LIN {X 0,Y 249.266,Z 167.431,A -85,B 0,C 180,E1 -18895.147,E2 -18895.147} C_VEL
LIN {X 0,Y 249.661,Z 167.386,A -85,B 0,C 180,E1 -18898.386,E2 -18898.386} C_VEL
LIN {X 0,Y 249.66,Z 167.377,A -85,B 0,C 180,E1 -18901.612,E2 -18901.612} C_VEL
LIN {X 0,Y 249.426,Z 167.411,A -85,B 0,C 180,E1 -18906.555,E2 -18906.555} C_VEL
LIN {X 0,Y 249.335,Z 167.427,A -85,B 0,C 180,E1 -18909.735,E2 -18909.735} C_VEL
LIN {X 0,Y 249.147,Z 167.433,A -85,B 0,C 180,E1 -18914.705,E2 -18914.705} C_VEL
LIN {X 0,Y 249.08,Z 167.45,A -85,B 0,C 180,E1 -18918.08,E2 -18918.08} C_VEL
LIN {X 0,Y 249.043,Z 167.464,A -85,B 0,C 180,E1 -18921.521,E2 -18921.521} C_VEL
LIN {X 0,Y 249.043,Z 167.454,A -85,B 0,C 180,E1 -18925.438,E2 -18925.438} C_VEL
LIN {X 0,Y 249.023,Z 167.452,A -85,B 0,C 180,E1 -18928.967,E2 -18928.967} C_VEL
LIN {X 0,Y 249.025,Z 167.464,A -85,B 0,C 180,E1 -18932.425,E2 -18932.425} C_VEL
LIN {X 0,Y 249.008,Z 167.459,A -85,B 0,C 180,E1 -18936.347,E2 -18936.347} C_VEL
LIN {X 0,Y 248.979,Z 167.466,A -85,B 0,C 180,E1 -18940.481,E2 -18940.481} C_VEL
LIN {X 0,Y 248.959,Z 167.473,A -85,B 0,C 180,E1 -18944.887,E2 -18944.887} C_VEL
LIN {X 0,Y 248.975,Z 167.462,A -85,B 0,C 180,E1 -18947.353,E2 -18947.353} C_VEL
LIN {X 0,Y 249.036,Z 167.465,A -85,B 0,C 180,E1 -18952.2,E2 -18952.2} C_VEL
LIN {X 0,Y 249.038,Z 167.459,A -85,B 0,C 180,E1 -18955.638,E2 -18955.638} C_VEL
LIN {X 0,Y 248.997,Z 167.467,A -85,B 0,C 180,E1 -18959.465,E2 -18959.465} C_VEL
LIN {X 0,Y 249.016,Z 167.467,A -85,B 0,C 180,E1 -18963.155,E2 -18963.155} C_VEL
LIN {X 0,Y 249,Z 167.461,A -85,B 0,C 180,E1 -18966.724,E2 -18966.724} C_VEL
LIN {X 0,Y 249.037,Z 167.466,A -85,B 0,C 180,E1 -18970.205,E2 -18970.205} C_VEL
LIN {X 0,Y 249.152,Z 167.449,A -85,B 0,C 180,E1 -18973.615,E2 -18973.615} C_VEL
LIN {X 0,Y 249.214,Z 167.439,A -85,B 0,C 180,E1 -18978.614,E2 -18978.614} C_VEL
LIN {X 0,Y 249.355,Z 167.424,A -85,B 0,C 180,E1 -18980.552,E2 -18980.552} C_VEL
LIN {X 0,Y 250.451,Z 170.4,A -85,B 0,C 180,E1 -18980.803,E2 -18980.803} C_VEL
LIN {X 0,Y 254.125,Z 177.882,A -85,B 0,C 180,E1 -18981.488,E2 -18981.488} C_VEL
LIN {X 0,Y 263.092,Z 200.069,A -85,B 0,C 180,E1 -18983.19,E2 -18983.19} C_VEL
LIN {X 0,Y 264.812,Z 205.047,A -85,B 0,C 180,E1 -18983.523,E2 -18983.523} C_VEL
LIN {X 0,Y 262.363,Z 274.189,A -85,B 0,C 180,E1 -18985.433,E2 -18985.433} C_VEL
LIN {X 0,Y 261.405,Z 287.63,A -85,B 0,C 180,E1 -18986.1,E2 -18986.1} C_VEL
LIN {X 0,Y 260.23,Z 300.609,A -85,B 0,C 180,E1 -18987.077,E2 -18987.077} C_VEL
LIN {X 0,Y 258.83,Z 312.038,A -85,B 0,C 180,E1 -18988.249,E2 -18988.249} C_VEL
LIN {X 0,Y 257.009,Z 323.786,A -85,B 0,C 180,E1 -18989.804,E2 -18989.804} C_VEL
LIN {X 0,Y 255.145,Z 334.352,A -85,B 0,C 180,E1 -18991.578,E2 -18991.578} C_VEL
LIN {X 0,Y 253.465,Z 343.314,A -85,B 0,C 180,E1 -18993.467,E2 -18993.467} C_VEL
LIN {X 0,Y 251.739,Z 351.564,A -85,B 0,C 180,E1 -18995.607,E2 -18995.607} C_VEL
LIN {X 0,Y 250.15,Z 359.176,A -85,B 0,C 180,E1 -18998.075,E2 -18998.075} C_VEL
LIN {X 0,Y 248.942,Z 365.251,A -85,B 0,C 180,E1 -19000.574,E2 -19000.574} C_VEL
LIN {X 0,Y 248.007,Z 370.011,A -85,B 0,C 180,E1 -19003.103,E2 -19003.103} C_VEL
LIN {X 0,Y 247.471,Z 372.881,A -85,B 0,C 180,E1 -19005.084,E2 -19005.084} C_VEL
LIN {X 0,Y 247.146,Z 374.563,A -85,B 0,C 180,E1 -19006.521,E2 -19006.521} C_VEL
LIN {X 0,Y 246.896,Z 376.129,A -85,B 0,C 180,E1 -19008.247,E2 -19008.247} C_VEL
LIN {X 0,Y 246.775,Z 377.22,A -85,B 0,C 180,E1 -19009.983,E2 -19009.983} C_VEL
LIN {X 0,Y 246.672,Z 377.893,A -85,B 0,C 180,E1 -19011.739,E2 -19011.739} C_VEL
LIN {X 0,Y 246.81,Z 378.021,A -85,B 0,C 180,E1 -19014.331,E2 -19014.331} C_VEL
LIN {X 0,Y 247.173,Z 377.088,A -85,B 0,C 180,E1 -19017.061,E2 -19017.061} C_VEL
LIN {X 0,Y 247.576,Z 375.846,A -85,B 0,C 180,E1 -19018.854,E2 -19018.854} C_VEL
LIN {X 0,Y 248.6,Z 372.467,A -85,B 0,C 180,E1 -19021.996,E2 -19021.996} C_VEL
LIN {X 0,Y 250.01,Z 367.842,A -85,B 0,C 180,E1 -19024.887,E2 -19024.887} C_VEL
LIN {X 0,Y 251.599,Z 362.394,A -85,B 0,C 180,E1 -19027.412,E2 -19027.412} C_VEL
LIN {X 0,Y 253.768,Z 354.935,A -85,B 0,C 180,E1 -19030.083,E2 -19030.083} C_VEL
LIN {X 0,Y 255.796,Z 347.755,A -85,B 0,C 180,E1 -19032.115,E2 -19032.115} C_VEL
LIN {X 0,Y 258.174,Z 338.472,A -85,B 0,C 180,E1 -19034.232,E2 -19034.232} C_VEL
LIN {X 0,Y 260.745,Z 327.432,A -85,B 0,C 180,E1 -19036.205,E2 -19036.205} C_VEL
LIN {X 0,Y 262.8,Z 317.371,A -85,B 0,C 180,E1 -19037.626,E2 -19037.626} C_VEL
LIN {X 0,Y 264.715,Z 306.116,A -85,B 0,C 180,E1 -19038.88,E2 -19038.88} C_VEL
LIN {X 0,Y 266.377,Z 293.716,A -85,B 0,C 180,E1 -19039.918,E2 -19039.918} C_VEL
LIN {X 0,Y 267.556,Z 280.481,A -85,B 0,C 180,E1 -19040.713,E2 -19040.713} C_VEL
LIN {X 0,Y 268.409,Z 267.04,A -85,B 0,C 180,E1 -19041.175,E2 -19041.175} C_VEL
LIN {X 0,Y 270.741,Z 210.533,A -85,B 0,C 180,E1 -19042.703,E2 -19042.703} C_VEL
LIN {X 0,Y 264.124,Z 195.268,A -85,B 0,C 180,E1 -19044.23,E2 -19044.23} C_VEL
LIN {X 0,Y 256.806,Z 181.169,A -85,B 0,C 180,E1 -19045.966,E2 -19045.966} C_VEL
LIN {X 0,Y 250.919,Z 171.414,A -85,B 0,C 180,E1 -19047.421,E2 -19047.421} C_VEL
LIN {X 0,Y 249.354,Z 168.806,A -85,B 0,C 180,E1 -19047.828,E2 -19047.828} C_VEL
LIN {X 0,Y 249.187,Z 168.189,A -85,B 0,C 180,E1 -19048.008,E2 -19048.008} C_VEL
LIN {X 0,Y 249.045,Z 167.461,A -85,B 0,C 180,E1 -19048.395,E2 -19048.395} C_VEL
LIN {X 0,Y 249.095,Z 167.458,A -85,B 0,C 180,E1 -19051.34,E2 -19051.34} C_VEL
LIN {X 0,Y 249.15,Z 167.451,A -85,B 0,C 180,E1 -19054.97,E2 -19054.97} C_VEL
LIN {X 0,Y 249.103,Z 167.456,A -85,B 0,C 180,E1 -19060.212,E2 -19060.212} C_VEL
LIN {X 0,Y 249.195,Z 167.44,A -85,B 0,C 180,E1 -19063.62,E2 -19063.62} C_VEL
LIN {X 0,Y 249.241,Z 167.438,A -85,B 0,C 180,E1 -19068.617,E2 -19068.617} C_VEL
LIN {X 0,Y 249.436,Z 167.403,A -85,B 0,C 180,E1 -19071.903,E2 -19071.903} C_VEL
LIN {X 0,Y 249.296,Z 167.415,A -85,B 0,C 180,E1 -19075.507,E2 -19075.507} C_VEL
LIN {X 0,Y 249.673,Z 167.382,A -85,B 0,C 180,E1 -19078.388,E2 -19078.388} C_VEL
LIN {X 0,Y 249.663,Z 167.37,A -85,B 0,C 180,E1 -19081.614,E2 -19081.614} C_VEL
LIN {X 0,Y 249.489,Z 167.394,A -85,B 0,C 180,E1 -19082.511,E2 -19082.511} C_VEL
LIN {X 0,Y 248.709,Z 167.502,A -85,B 0,C 180,E1 -19083.857,E2 -19083.857} C_VEL
LIN {X 0,Y 245.911,Z 167.861,A -85,B 0,C 180,E1 -19086.056,E2 -19086.056} C_VEL
LIN {X 0,Y 242.72,Z 168.25,A -85,B 0,C 180,E1 -19088.763,E2 -19088.763} C_VEL
LIN {X 0,Y 242.313,Z 168.291,A -85,B 0,C 180,E1 -19089.698,E2 -19089.698} C_VEL
LIN {X 0,Y 242.119,Z 168.317,A -85,B 0,C 180,E1 -19095.145,E2 -19095.145} C_VEL
LIN {X 0,Y 242.031,Z 168.337,A -85,B 0,C 180,E1 -19098.629,E2 -19098.629} C_VEL
LIN {X 0,Y 241.975,Z 168.332,A -85,B 0,C 180,E1 -19102.185,E2 -19102.185} C_VEL
LIN {X 0,Y 241.989,Z 168.329,A -85,B 0,C 180,E1 -19105.827,E2 -19105.827} C_VEL
LIN {X 0,Y 241.971,Z 168.337,A -85,B 0,C 180,E1 -19109.59,E2 -19109.59} C_VEL
LIN {X 0,Y 241.982,Z 168.338,A -85,B 0,C 180,E1 -19113.494,E2 -19113.494} C_VEL
LIN {X 0,Y 241.967,Z 168.338,A -85,B 0,C 180,E1 -19117.587,E2 -19117.587} C_VEL
LIN {X 0,Y 241.907,Z 168.352,A -85,B 0,C 180,E1 -19121.93,E2 -19121.93} C_VEL
LIN {X 0,Y 241.902,Z 168.356,A -85,B 0,C 180,E1 -19126.581,E2 -19126.581} C_VEL
LIN {X 0,Y 241.927,Z 168.36,A -85,B 0,C 180,E1 -19127.022,E2 -19127.022} C_VEL
LIN {X 0,Y 244.494,Z 177.241,A -85,B 0,C 180,E1 -19131.493,E2 -19131.493} C_VEL
LIN {X 0,Y 245.657,Z 181.596,A -85,B 0,C 180,E1 -19133.461,E2 -19133.461} C_VEL
LIN {X 0,Y 248.1,Z 186.109,A -85,B 0,C 180,E1 -19134.124,E2 -19134.124} C_VEL
LIN {X 0,Y 254.965,Z 199.897,A -85,B 0,C 180,E1 -19135.919,E2 -19135.919} C_VEL
LIN {X 0,Y 260.527,Z 212.758,A -85,B 0,C 180,E1 -19137.324,E2 -19137.324} C_VEL
LIN {X 0,Y 263.753,Z 235.456,A -85,B 0,C 180,E1 -19138.613,E2 -19138.613} C_VEL
LIN {X 0,Y 263.05,Z 257.778,A -85,B 0,C 180,E1 -19139.265,E2 -19139.265} C_VEL
LIN {X 0,Y 261.59,Z 291.145,A -85,B 0,C 180,E1 -19140.226,E2 -19140.226} C_VEL
LIN {X 0,Y 260.253,Z 304.533,A -85,B 0,C 180,E1 -19140.869,E2 -19140.869} C_VEL
LIN {X 0,Y 258.368,Z 317.473,A -85,B 0,C 180,E1 -19141.795,E2 -19141.795} C_VEL
LIN {X 0,Y 256.335,Z 328.522,A -85,B 0,C 180,E1 -19142.883,E2 -19142.883} C_VEL
LIN {X 0,Y 253.936,Z 340.052,A -85,B 0,C 180,E1 -19144.378,E2 -19144.378} C_VEL
LIN {X 0,Y 251.38,Z 350.474,A -85,B 0,C 180,E1 -19146.085,E2 -19146.085} C_VEL
LIN {X 0,Y 248.823,Z 359.904,A -85,B 0,C 180,E1 -19148.022,E2 -19148.022} C_VEL
LIN {X 0,Y 246.406,Z 369.146,A -85,B 0,C 180,E1 -19150.459,E2 -19150.459} C_VEL
LIN {X 0,Y 244.321,Z 376.399,A -85,B 0,C 180,E1 -19152.852,E2 -19152.852} C_VEL
LIN {X 0,Y 242.243,Z 383.198,A -85,B 0,C 180,E1 -19155.724,E2 -19155.724} C_VEL
LIN {X 0,Y 241.112,Z 387.712,A -85,B 0,C 180,E1 -19158.227,E2 -19158.227} C_VEL
LIN {X 0,Y 240.55,Z 390.106,A -85,B 0,C 180,E1 -19159.904,E2 -19159.904} C_VEL
LIN {X 0,Y 240.167,Z 392.075,A -85,B 0,C 180,E1 -19161.587,E2 -19161.587} C_VEL
LIN {X 0,Y 239.904,Z 393.622,A -85,B 0,C 180,E1 -19163.271,E2 -19163.271} C_VEL
LIN {X 0,Y 239.783,Z 394.866,A -85,B 0,C 180,E1 -19165.241,E2 -19165.241} C_VEL
LIN {X 0,Y 239.885,Z 395.756,A -85,B 0,C 180,E1 -19168.321,E2 -19168.321} C_VEL
LIN {X 0,Y 239.959,Z 395.682,A -85,B 0,C 180,E1 -19170,E2 -19170} C_VEL
LIN {X 0,Y 239.912,Z 395.161,A -85,B 0,C 180,E1 -19171.679,E2 -19171.679} C_VEL
LIN {X 0,Y 239.786,Z 393.146,A -85,B 0,C 180,E1 -19174.767,E2 -19174.767} C_VEL
LIN {X 0,Y 240.029,Z 390.076,A -85,B 0,C 180,E1 -19177.572,E2 -19177.572} C_VEL
LIN {X 0,Y 240.501,Z 386.195,A -85,B 0,C 180,E1 -19180.098,E2 -19180.098} C_VEL
LIN {X 0,Y 241.269,Z 381.159,A -85,B 0,C 180,E1 -19182.62,E2 -19182.62} C_VEL
LIN {X 0,Y 242.591,Z 374.83,A -85,B 0,C 180,E1 -19185.114,E2 -19185.114} C_VEL
LIN {X 0,Y 244.27,Z 366.88,A -85,B 0,C 180,E1 -19187.584,E2 -19187.584} C_VEL
LIN {X 0,Y 245.795,Z 358.736,A -85,B 0,C 180,E1 -19189.634,E2 -19189.634} C_VEL
LIN {X 0,Y 247.688,Z 348.828,A -85,B 0,C 180,E1 -19191.646,E2 -19191.646} C_VEL
LIN {X 0,Y 249.586,Z 339.115,A -85,B 0,C 180,E1 -19193.218,E2 -19193.218} C_VEL
LIN {X 0,Y 251.397,Z 328.643,A -85,B 0,C 180,E1 -19194.573,E2 -19194.573} C_VEL
LIN {X 0,Y 253.211,Z 316.059,A -85,B 0,C 180,E1 -19195.812,E2 -19195.812} C_VEL
LIN {X 0,Y 254.709,Z 302.824,A -85,B 0,C 180,E1 -19196.751,E2 -19196.751} C_VEL
LIN {X 0,Y 255.579,Z 290.802,A -85,B 0,C 180,E1 -19197.315,E2 -19197.315} C_VEL
LIN {X 0,Y 257.476,Z 234.096,A -85,B 0,C 180,E1 -19198.933,E2 -19198.933} C_VEL
LIN {X 0,Y 253.141,Z 203.077,A -85,B 0,C 180,E1 -19200.402,E2 -19200.402} C_VEL
LIN {X 0,Y 246.374,Z 185.846,A -85,B 0,C 180,E1 -19201.778,E2 -19201.778} C_VEL
LIN {X 0,Y 245.337,Z 183.037,A -85,B 0,C 180,E1 -19202.03,E2 -19202.03} C_VEL
LIN {X 0,Y 243.166,Z 173.071,A -85,B 0,C 180,E1 -19205.975,E2 -19205.975} C_VEL
LIN {X 0,Y 241.972,Z 168.341,A -85,B 0,C 180,E1 -19207.969,E2 -19207.969} C_VEL
LIN {X 0,Y 241.904,Z 168.344,A -85,B 0,C 180,E1 -19211.93,E2 -19211.93} C_VEL
LIN {X 0,Y 241.905,Z 168.352,A -85,B 0,C 180,E1 -19216.579,E2 -19216.579} C_VEL
LIN {X 0,Y 241.998,Z 168.343,A -85,B 0,C 180,E1 -19221.641,E2 -19221.641} C_VEL
LIN {X 0,Y 241.985,Z 168.344,A -85,B 0,C 180,E1 -19224.487,E2 -19224.487} C_VEL
LIN {X 0,Y 241.958,Z 168.346,A -85,B 0,C 180,E1 -19228.476,E2 -19228.476} C_VEL
LIN {X 0,Y 241.973,Z 168.344,A -85,B 0,C 180,E1 -19232.307,E2 -19232.307} C_VEL
LIN {X 0,Y 242.028,Z 168.336,A -85,B 0,C 180,E1 -19236.012,E2 -19236.012} C_VEL
LIN {X 0,Y 241.99,Z 168.339,A -85,B 0,C 180,E1 -19239.602,E2 -19239.602} C_VEL
LIN {X 0,Y 242.11,Z 168.325,A -85,B 0,C 180,E1 -19243.323,E2 -19243.323} C_VEL
LIN {X 0,Y 242.166,Z 168.319,A -85,B 0,C 180,E1 -19248.277,E2 -19248.277} C_VEL
LIN {X 0,Y 242.376,Z 168.276,A -85,B 0,C 180,E1 -19251.662,E2 -19251.662} C_VEL
LIN {X 0,Y 242.401,Z 168.278,A -85,B 0,C 180,E1 -19253.339,E2 -19253.339} C_VEL
LIN {X 0,Y 242.621,Z 168.263,A -85,B 0,C 180,E1 -19258.339,E2 -19258.339} C_VEL
LIN {X 0,Y 242.62,Z 168.252,A -85,B 0,C 180,E1 -19261.659,E2 -19261.659} C_VEL
LIN {X 0,Y 242.402,Z 168.286,A -85,B 0,C 180,E1 -19266.658,E2 -19266.658} C_VEL
LIN {X 0,Y 242.262,Z 168.309,A -85,B 0,C 180,E1 -19270.022,E2 -19270.022} C_VEL
LIN {X 0,Y 242.105,Z 168.308,A -85,B 0,C 180,E1 -19275.143,E2 -19275.143} C_VEL
LIN {X 0,Y 242.018,Z 168.331,A -85,B 0,C 180,E1 -19278.627,E2 -19278.627} C_VEL
LIN {X 0,Y 241.973,Z 168.343,A -85,B 0,C 180,E1 -19282.182,E2 -19282.182} C_VEL
LIN {X 0,Y 241.986,Z 168.328,A -85,B 0,C 180,E1 -19285.825,E2 -19285.825} C_VEL
LIN {X 0,Y 241.962,Z 168.335,A -85,B 0,C 180,E1 -19289.588,E2 -19289.588} C_VEL
LIN {X 0,Y 241.977,Z 168.344,A -85,B 0,C 180,E1 -19293.491,E2 -19293.491} C_VEL
LIN {X 0,Y 241.963,Z 168.329,A -85,B 0,C 180,E1 -19297.585,E2 -19297.585} C_VEL
LIN {X 0,Y 241.906,Z 168.352,A -85,B 0,C 180,E1 -19301.927,E2 -19301.927} C_VEL
LIN {X 0,Y 241.897,Z 168.345,A -85,B 0,C 180,E1 -19306.578,E2 -19306.578} C_VEL
LIN {X 0,Y 241.988,Z 168.343,A -85,B 0,C 180,E1 -19311.64,E2 -19311.64} C_VEL
LIN {X 0,Y 241.975,Z 168.338,A -85,B 0,C 180,E1 -19314.486,E2 -19314.486} C_VEL
LIN {X 0,Y 241.948,Z 168.349,A -85,B 0,C 180,E1 -19318.475,E2 -19318.475} C_VEL
LIN {X 0,Y 241.955,Z 168.341,A -85,B 0,C 180,E1 -19322.306,E2 -19322.306} C_VEL
LIN {X 0,Y 241.976,Z 168.338,A -85,B 0,C 180,E1 -19326.007,E2 -19326.007} C_VEL
LIN {X 0,Y 241.977,Z 168.344,A -85,B 0,C 180,E1 -19329.602,E2 -19329.602} C_VEL
LIN {X 0,Y 242.099,Z 168.327,A -85,B 0,C 180,E1 -19333.324,E2 -19333.324} C_VEL
LIN {X 0,Y 242.148,Z 168.32,A -85,B 0,C 180,E1 -19338.278,E2 -19338.278} C_VEL
LIN {X 0,Y 242.223,Z 168.31,A -85,B 0,C 180,E1 -19339.671,E2 -19339.671} C_VEL
LIN {X 0,Y 243.295,Z 171.211,A -85,B 0,C 180,E1 -19339.937,E2 -19339.937} C_VEL
LIN {X 0,Y 247.992,Z 180.283,A -85,B 0,C 180,E1 -19340.833,E2 -19340.833} C_VEL
LIN {X 0,Y 257.163,Z 203.11,A -85,B 0,C 180,E1 -19342.648,E2 -19342.648} C_VEL
LIN {X 0,Y 258.309,Z 206.449,A -85,B 0,C 180,E1 -19342.879,E2 -19342.879} C_VEL
LIN {X 0,Y 256.752,Z 251.318,A -85,B 0,C 180,E1 -19344.13,E2 -19344.13} C_VEL
LIN {X 0,Y 255.797,Z 275.757,A -85,B 0,C 180,E1 -19344.864,E2 -19344.864} C_VEL
LIN {X 0,Y 254.746,Z 289.229,A -85,B 0,C 180,E1 -19345.573,E2 -19345.573} C_VEL
LIN {X 0,Y 253.611,Z 301.204,A -85,B 0,C 180,E1 -19346.52,E2 -19346.52} C_VEL
LIN {X 0,Y 252.045,Z 313.242,A -85,B 0,C 180,E1 -19347.802,E2 -19347.802} C_VEL
LIN {X 0,Y 250.189,Z 324.811,A -85,B 0,C 180,E1 -19349.396,E2 -19349.396} C_VEL
LIN {X 0,Y 248.269,Z 335.207,A -85,B 0,C 180,E1 -19351.216,E2 -19351.216} C_VEL
LIN {X 0,Y 246.384,Z 344.7,A -85,B 0,C 180,E1 -19353.31,E2 -19353.31} C_VEL
LIN {X 0,Y 244.493,Z 353.629,A -85,B 0,C 180,E1 -19355.774,E2 -19355.774} C_VEL
LIN {X 0,Y 242.877,Z 360.869,A -85,B 0,C 180,E1 -19358.319,E2 -19358.319} C_VEL
LIN {X 0,Y 241.685,Z 366.622,A -85,B 0,C 180,E1 -19360.895,E2 -19360.895} C_VEL
LIN {X 0,Y 240.792,Z 371.122,A -85,B 0,C 180,E1 -19363.503,E2 -19363.503} C_VEL
LIN {X 0,Y 240.328,Z 373.508,A -85,B 0,C 180,E1 -19365.259,E2 -19365.259} C_VEL
LIN {X 0,Y 239.967,Z 375.378,A -85,B 0,C 180,E1 -19367.03,E2 -19367.03} C_VEL
LIN {X 0,Y 239.677,Z 377.585,A -85,B 0,C 180,E1 -19370.232,E2 -19370.232} C_VEL
LIN {X 0,Y 239.579,Z 378.26,A -85,B 0,C 180,E1 -19372.417,E2 -19372.417} C_VEL
LIN {X 0,Y 239.742,Z 378.269,A -85,B 0,C 180,E1 -19374.67,E2 -19374.67} C_VEL
LIN {X 0,Y 240.272,Z 376.991,A -85,B 0,C 180,E1 -19377.905,E2 -19377.905} C_VEL
LIN {X 0,Y 240.73,Z 375.602,A -85,B 0,C 180,E1 -19379.756,E2 -19379.756} C_VEL
LIN {X 0,Y 241.702,Z 372.565,A -85,B 0,C 180,E1 -19382.52,E2 -19382.52} C_VEL
LIN {X 0,Y 243.151,Z 368.181,A -85,B 0,C 180,E1 -19385.315,E2 -19385.315} C_VEL
LIN {X 0,Y 244.939,Z 362.315,A -85,B 0,C 180,E1 -19388.09,E2 -19388.09} C_VEL
LIN {X 0,Y 247.262,Z 354.78,A -85,B 0,C 180,E1 -19390.824,E2 -19390.824} C_VEL
LIN {X 0,Y 249.64,Z 346.693,A -85,B 0,C 180,E1 -19393.107,E2 -19393.107} C_VEL
LIN {X 0,Y 252.24,Z 337.015,A -85,B 0,C 180,E1 -19395.275,E2 -19395.275} C_VEL
LIN {X 0,Y 254.552,Z 327.254,A -85,B 0,C 180,E1 -19397.024,E2 -19397.024} C_VEL
LIN {X 0,Y 256.695,Z 317.246,A -85,B 0,C 180,E1 -19398.453,E2 -19398.453} C_VEL
LIN {X 0,Y 258.805,Z 305.163,A -85,B 0,C 180,E1 -19399.796,E2 -19399.796} C_VEL
LIN {X 0,Y 260.518,Z 292.361,A -85,B 0,C 180,E1 -19400.858,E2 -19400.858} C_VEL
LIN {X 0,Y 261.712,Z 279.403,A -85,B 0,C 180,E1 -19401.602,E2 -19401.602} C_VEL
LIN {X 0,Y 262.647,Z 263.353,A -85,B 0,C 180,E1 -19402.124,E2 -19402.124} C_VEL
LIN {X 0,Y 264.753,Z 212.279,A -85,B 0,C 180,E1 -19403.546,E2 -19403.546} C_VEL
LIN {X 0,Y 258.632,Z 198.245,A -85,B 0,C 180,E1 -19405.028,E2 -19405.028} C_VEL
LIN {X 0,Y 252.104,Z 185.543,A -85,B 0,C 180,E1 -19406.655,E2 -19406.655} C_VEL
LIN {X 0,Y 246.497,Z 176.218,A -85,B 0,C 180,E1 -19408.103,E2 -19408.103} C_VEL
LIN {X 0,Y 244.36,Z 172.777,A -85,B 0,C 180,E1 -19408.682,E2 -19408.682} C_VEL
LIN {X 0,Y 242.54,Z 170.296,A -85,B 0,C 180,E1 -19409.17,E2 -19409.17} C_VEL
LIN {X 0,Y 242.079,Z 168.811,A -85,B 0,C 180,E1 -19409.346,E2 -19409.346} C_VEL
LIN {X 0,Y 242.013,Z 168.338,A -85,B 0,C 180,E1 -19409.699,E2 -19409.699} C_VEL
LIN {X 0,Y 242.066,Z 168.337,A -85,B 0,C 180,E1 -19414.184,E2 -19414.184} C_VEL
LIN {X 0,Y 242.052,Z 168.332,A -85,B 0,C 180,E1 -19418.299,E2 -19418.299} C_VEL
LIN {X 0,Y 242.154,Z 168.315,A -85,B 0,C 180,E1 -19423.287,E2 -19423.287} C_VEL
LIN {X 0,Y 242.177,Z 168.317,A -85,B 0,C 180,E1 -19428.281,E2 -19428.281} C_VEL
LIN {X 0,Y 242.386,Z 168.28,A -85,B 0,C 180,E1 -19431.666,E2 -19431.666} C_VEL
LIN {X 0,Y 242.241,Z 168.297,A -85,B 0,C 180,E1 -19435.008,E2 -19435.008} C_VEL
LIN {X 0,Y 242.633,Z 168.259,A -85,B 0,C 180,E1 -19438.342,E2 -19438.342} C_VEL
LIN {X 0,Y 242.622,Z 168.247,A -85,B 0,C 180,E1 -19441.661,E2 -19441.661} C_VEL
LIN {X 0,Y 242.403,Z 168.273,A -85,B 0,C 180,E1 -19446.661,E2 -19446.661} C_VEL
LIN {X 0,Y 242.313,Z 168.291,A -85,B 0,C 180,E1 -19449.698,E2 -19449.698} C_VEL
LIN {X 0,Y 241.514,Z 168.386,A -85,B 0,C 180,E1 -19451.083,E2 -19451.083} C_VEL
LIN {X 0,Y 238.636,Z 168.758,A -85,B 0,C 180,E1 -19453.342,E2 -19453.342} C_VEL
LIN {X 0,Y 235.41,Z 169.146,A -85,B 0,C 180,E1 -19456.127,E2 -19456.127} C_VEL
LIN {X 0,Y 235.038,Z 169.194,A -85,B 0,C 180,E1 -19457.091,E2 -19457.091} C_VEL
LIN {X 0,Y 234.96,Z 169.204,A -85,B 0,C 180,E1 -19461.989,E2 -19461.989} C_VEL
LIN {X 0,Y 234.928,Z 169.209,A -85,B 0,C 180,E1 -19466.664,E2 -19466.664} C_VEL
LIN {X 0,Y 234.901,Z 169.213,A -85,B 0,C 180,E1 -19470.574,E2 -19470.574} C_VEL
LIN {X 0,Y 234.924,Z 169.212,A -85,B 0,C 180,E1 -19474.64,E2 -19474.64} C_VEL
LIN {X 0,Y 234.914,Z 169.22,A -85,B 0,C 180,E1 -19478.936,E2 -19478.936} C_VEL
LIN {X 0,Y 234.855,Z 169.233,A -85,B 0,C 180,E1 -19483.495,E2 -19483.495} C_VEL
LIN {X 0,Y 234.882,Z 169.447,A -85,B 0,C 180,E1 -19485.777,E2 -19485.777} C_VEL
LIN {X 0,Y 236.957,Z 176.353,A -85,B 0,C 180,E1 -19489.516,E2 -19489.516} C_VEL
LIN {X 0,Y 238.318,Z 181.118,A -85,B 0,C 180,E1 -19491.88,E2 -19491.88} C_VEL
LIN {X 0,Y 240.737,Z 185.589,A -85,B 0,C 180,E1 -19492.598,E2 -19492.598} C_VEL
LIN {X 0,Y 246.246,Z 195.927,A -85,B 0,C 180,E1 -19494.147,E2 -19494.147} C_VEL
LIN {X 0,Y 252.545,Z 209.432,A -85,B 0,C 180,E1 -19495.842,E2 -19495.842} C_VEL
LIN {X 0,Y 255.206,Z 216.173,A -85,B 0,C 180,E1 -19496.557,E2 -19496.557} C_VEL
LIN {X 0,Y 258.041,Z 237.547,A -85,B 0,C 180,E1 -19497.796,E2 -19497.796} C_VEL
LIN {X 0,Y 255.66,Z 291.409,A -85,B 0,C 180,E1 -19499.369,E2 -19499.369} C_VEL
LIN {X 0,Y 254.196,Z 305.151,A -85,B 0,C 180,E1 -19500.052,E2 -19500.052} C_VEL
LIN {X 0,Y 252.36,Z 317.268,A -85,B 0,C 180,E1 -19500.947,E2 -19500.947} C_VEL
LIN {X 0,Y 250.069,Z 329.087,A -85,B 0,C 180,E1 -19502.145,E2 -19502.145} C_VEL
LIN {X 0,Y 247.577,Z 340.468,A -85,B 0,C 180,E1 -19503.67,E2 -19503.67} C_VEL
LIN {X 0,Y 244.919,Z 350.774,A -85,B 0,C 180,E1 -19505.413,E2 -19505.413} C_VEL
LIN {X 0,Y 242.256,Z 360.065,A -85,B 0,C 180,E1 -19507.394,E2 -19507.394} C_VEL
LIN {X 0,Y 239.887,Z 368.414,A -85,B 0,C 180,E1 -19509.641,E2 -19509.641} C_VEL
LIN {X 0,Y 237.513,Z 376.402,A -85,B 0,C 180,E1 -19512.345,E2 -19512.345} C_VEL
LIN {X 0,Y 235.35,Z 383.124,A -85,B 0,C 180,E1 -19515.296,E2 -19515.296} C_VEL
LIN {X 0,Y 234.127,Z 387.594,A -85,B 0,C 180,E1 -19517.871,E2 -19517.871} C_VEL
LIN {X 0,Y 233.533,Z 389.969,A -85,B 0,C 180,E1 -19519.598,E2 -19519.598} C_VEL
LIN {X 0,Y 233.114,Z 391.918,A -85,B 0,C 180,E1 -19521.33,E2 -19521.33} C_VEL
LIN {X 0,Y 232.826,Z 393.429,A -85,B 0,C 180,E1 -19523.065,E2 -19523.065} C_VEL
LIN {X 0,Y 232.702,Z 394.765,A -85,B 0,C 180,E1 -19525.326,E2 -19525.326} C_VEL
LIN {X 0,Y 232.794,Z 395.505,A -85,B 0,C 180,E1 -19528.27,E2 -19528.27} C_VEL
LIN {X 0,Y 232.889,Z 395.4,A -85,B 0,C 180,E1 -19530,E2 -19530} C_VEL
LIN {X 0,Y 232.819,Z 394.853,A -85,B 0,C 180,E1 -19531.73,E2 -19531.73} C_VEL
LIN {X 0,Y 232.707,Z 392.988,A -85,B 0,C 180,E1 -19534.688,E2 -19534.688} C_VEL
LIN {X 0,Y 232.983,Z 389.687,A -85,B 0,C 180,E1 -19537.802,E2 -19537.802} C_VEL
LIN {X 0,Y 233.48,Z 385.76,A -85,B 0,C 180,E1 -19540.406,E2 -19540.406} C_VEL
LIN {X 0,Y 234.303,Z 380.676,A -85,B 0,C 180,E1 -19543.001,E2 -19543.001} C_VEL
LIN {X 0,Y 235.723,Z 374.283,A -85,B 0,C 180,E1 -19545.565,E2 -19545.565} C_VEL
LIN {X 0,Y 237.445,Z 366.25,A -85,B 0,C 180,E1 -19548.107,E2 -19548.107} C_VEL
LIN {X 0,Y 239.048,Z 358.044,A -85,B 0,C 180,E1 -19550.209,E2 -19550.209} C_VEL
LIN {X 0,Y 241.111,Z 348.044,A -85,B 0,C 180,E1 -19552.268,E2 -19552.268} C_VEL
LIN {X 0,Y 243.312,Z 336.781,A -85,B 0,C 180,E1 -19554.08,E2 -19554.08} C_VEL
LIN {X 0,Y 245.224,Z 325.752,A -85,B 0,C 180,E1 -19555.461,E2 -19555.461} C_VEL
LIN {X 0,Y 247.008,Z 313.567,A -85,B 0,C 180,E1 -19556.624,E2 -19556.624} C_VEL
LIN {X 0,Y 248.338,Z 300.863,A -85,B 0,C 180,E1 -19557.494,E2 -19557.494} C_VEL
LIN {X 0,Y 249.232,Z 287.638,A -85,B 0,C 180,E1 -19558.071,E2 -19558.071} C_VEL
LIN {X 0,Y 250.999,Z 234.479,A -85,B 0,C 180,E1 -19559.619,E2 -19559.619} C_VEL
LIN {X 0,Y 246.863,Z 204.961,A -85,B 0,C 180,E1 -19561.074,E2 -19561.074} C_VEL
LIN {X 0,Y 239.328,Z 186.004,A -85,B 0,C 180,E1 -19562.667,E2 -19562.667} C_VEL
LIN {X 0,Y 238.077,Z 182.749,A -85,B 0,C 180,E1 -19562.979,E2 -19562.979} C_VEL
LIN {X 0,Y 236.15,Z 174.109,A -85,B 0,C 180,E1 -19566.529,E2 -19566.529} C_VEL
LIN {X 0,Y 234.913,Z 169.218,A -85,B 0,C 180,E1 -19568.648,E2 -19568.648} C_VEL
LIN {X 0,Y 234.851,Z 169.226,A -85,B 0,C 180,E1 -19573.495,E2 -19573.495} C_VEL
LIN {X 0,Y 234.858,Z 169.23,A -85,B 0,C 180,E1 -19576.506,E2 -19576.506} C_VEL
LIN {X 0,Y 234.923,Z 169.225,A -85,B 0,C 180,E1 -19581.078,E2 -19581.078} C_VEL
LIN {X 0,Y 234.931,Z 169.223,A -85,B 0,C 180,E1 -19585.361,E2 -19585.361} C_VEL
LIN {X 0,Y 234.904,Z 169.225,A -85,B 0,C 180,E1 -19589.427,E2 -19589.427} C_VEL
LIN {X 0,Y 234.974,Z 169.215,A -85,B 0,C 180,E1 -19593.806,E2 -19593.806} C_VEL
LIN {X 0,Y 234.97,Z 169.215,A -85,B 0,C 180,E1 -19598.007,E2 -19598.007} C_VEL
LIN {X 0,Y 235.054,Z 169.205,A -85,B 0,C 180,E1 -19603.097,E2 -19603.097} C_VEL
LIN {X 0,Y 235.096,Z 169.199,A -85,B 0,C 180,E1 -19607.92,E2 -19607.92} C_VEL
LIN {X 0,Y 235.315,Z 169.155,A -85,B 0,C 180,E1 -19611.41,E2 -19611.41} C_VEL
LIN {X 0,Y 235.352,Z 169.155,A -85,B 0,C 180,E1 -19613.138,E2 -19613.138} C_VEL
LIN {X 0,Y 235.58,Z 169.141,A -85,B 0,C 180,E1 -19618.289,E2 -19618.289} C_VEL
LIN {X 0,Y 235.579,Z 169.127,A -85,B 0,C 180,E1 -19621.708,E2 -19621.708} C_VEL
LIN {X 0,Y 235.354,Z 169.163,A -85,B 0,C 180,E1 -19626.859,E2 -19626.859} C_VEL
LIN {X 0,Y 235.186,Z 169.188,A -85,B 0,C 180,E1 -19630.327,E2 -19630.327} C_VEL
LIN {X 0,Y 235.042,Z 169.185,A -85,B 0,C 180,E1 -19635.61,E2 -19635.61} C_VEL
LIN {X 0,Y 234.959,Z 169.211,A -85,B 0,C 180,E1 -19639.208,E2 -19639.208} C_VEL
LIN {X 0,Y 234.908,Z 169.222,A -85,B 0,C 180,E1 -19642.887,E2 -19642.887} C_VEL
LIN {X 0,Y 234.921,Z 169.205,A -85,B 0,C 180,E1 -19646.662,E2 -19646.662} C_VEL
LIN {X 0,Y 234.894,Z 169.22,A -85,B 0,C 180,E1 -19650.571,E2 -19650.571} C_VEL
LIN {X 0,Y 234.92,Z 169.22,A -85,B 0,C 180,E1 -19654.638,E2 -19654.638} C_VEL
LIN {X 0,Y 234.909,Z 169.208,A -85,B 0,C 180,E1 -19658.933,E2 -19658.933} C_VEL
LIN {X 0,Y 234.85,Z 169.232,A -85,B 0,C 180,E1 -19663.492,E2 -19663.492} C_VEL
LIN {X 0,Y 234.849,Z 169.222,A -85,B 0,C 180,E1 -19666.504,E2 -19666.504} C_VEL
LIN {X 0,Y 234.914,Z 169.228,A -85,B 0,C 180,E1 -19671.077,E2 -19671.077} C_VEL
LIN {X 0,Y 234.921,Z 169.215,A -85,B 0,C 180,E1 -19675.36,E2 -19675.36} C_VEL
LIN {X 0,Y 234.894,Z 169.224,A -85,B 0,C 180,E1 -19679.426,E2 -19679.426} C_VEL
LIN {X 0,Y 234.935,Z 169.22,A -85,B 0,C 180,E1 -19683.819,E2 -19683.819} C_VEL
LIN {X 0,Y 234.93,Z 169.223,A -85,B 0,C 180,E1 -19688.962,E2 -19688.962} C_VEL
LIN {X 0,Y 235.043,Z 169.206,A -85,B 0,C 180,E1 -19693.097,E2 -19693.097} C_VEL
LIN {X 0,Y 235.08,Z 169.203,A -85,B 0,C 180,E1 -19697.92,E2 -19697.92} C_VEL
LIN {X 0,Y 235.142,Z 169.19,A -85,B 0,C 180,E1 -19698.753,E2 -19698.753} C_VEL
LIN {X 0,Y 236.233,Z 172.126,A -85,B 0,C 180,E1 -19699.03,E2 -19699.03} C_VEL
LIN {X 0,Y 241.596,Z 182.194,A -85,B 0,C 180,E1 -19700.097,E2 -19700.097} C_VEL
LIN {X 0,Y 250.799,Z 204.797,A -85,B 0,C 180,E1 -19701.983,E2 -19701.983} C_VEL
LIN {X 0,Y 251.948,Z 208.231,A -85,B 0,C 180,E1 -19702.228,E2 -19702.228} C_VEL
LIN {X 0,Y 249.361,Z 275.351,A -85,B 0,C 180,E1 -19704.179,E2 -19704.179} C_VEL
LIN {X 0,Y 248.314,Z 288.724,A -85,B 0,C 180,E1 -19704.885,E2 -19704.885} C_VEL
LIN {X 0,Y 247.072,Z 301.28,A -85,B 0,C 180,E1 -19705.885,E2 -19705.885} C_VEL
LIN {X 0,Y 245.567,Z 312.786,A -85,B 0,C 180,E1 -19707.129,E2 -19707.129} C_VEL
LIN {X 0,Y 243.611,Z 324.496,A -85,B 0,C 180,E1 -19708.76,E2 -19708.76} C_VEL
LIN {X 0,Y 241.617,Z 335.021,A -85,B 0,C 180,E1 -19710.625,E2 -19710.625} C_VEL
LIN {X 0,Y 239.516,Z 345.128,A -85,B 0,C 180,E1 -19712.907,E2 -19712.907} C_VEL
LIN {X 0,Y 237.787,Z 352.891,A -85,B 0,C 180,E1 -19715.087,E2 -19715.087} C_VEL
LIN {X 0,Y 236.083,Z 360.368,A -85,B 0,C 180,E1 -19717.698,E2 -19717.698} C_VEL
LIN {X 0,Y 234.81,Z 366.276,A -85,B 0,C 180,E1 -19720.345,E2 -19720.345} C_VEL
LIN {X 0,Y 233.838,Z 370.913,A -85,B 0,C 180,E1 -19723.027,E2 -19723.027} C_VEL
LIN {X 0,Y 233.102,Z 374.41,A -85,B 0,C 180,E1 -19725.744,E2 -19725.744} C_VEL
LIN {X 0,Y 232.793,Z 376.141,A -85,B 0,C 180,E1 -19727.571,E2 -19727.571} C_VEL
LIN {X 0,Y 232.545,Z 377.938,A -85,B 0,C 180,E1 -19730.47,E2 -19730.47} C_VEL
LIN {X 0,Y 232.513,Z 378.588,A -85,B 0,C 180,E1 -19733.137,E2 -19733.137} C_VEL
LIN {X 0,Y 232.695,Z 378.5,A -85,B 0,C 180,E1 -19735.035,E2 -19735.035} C_VEL
LIN {X 0,Y 232.965,Z 377.91,A -85,B 0,C 180,E1 -19736.905,E2 -19736.905} C_VEL
LIN {X 0,Y 233.492,Z 376.588,A -85,B 0,C 180,E1 -19739.208,E2 -19739.208} C_VEL
LIN {X 0,Y 234.266,Z 374.34,A -85,B 0,C 180,E1 -19741.668,E2 -19741.668} C_VEL
LIN {X 0,Y 235.551,Z 370.573,A -85,B 0,C 180,E1 -19744.534,E2 -19744.534} C_VEL
LIN {X 0,Y 237.365,Z 365.21,A -85,B 0,C 180,E1 -19747.478,E2 -19747.478} C_VEL
LIN {X 0,Y 239.589,Z 358.435,A -85,B 0,C 180,E1 -19750.302,E2 -19750.302} C_VEL
LIN {X 0,Y 241.758,Z 351.646,A -85,B 0,C 180,E1 -19752.523,E2 -19752.523} C_VEL
LIN {X 0,Y 244.342,Z 342.917,A -85,B 0,C 180,E1 -19754.805,E2 -19754.805} C_VEL
LIN {X 0,Y 247.191,Z 332.361,A -85,B 0,C 180,E1 -19756.974,E2 -19756.974} C_VEL
LIN {X 0,Y 249.499,Z 322.475,A -85,B 0,C 180,E1 -19758.589,E2 -19758.589} C_VEL
LIN {X 0,Y 251.668,Z 312.256,A -85,B 0,C 180,E1 -19759.902,E2 -19759.902} C_VEL
LIN {X 0,Y 253.507,Z 300.703,A -85,B 0,C 180,E1 -19761.076,E2 -19761.076} C_VEL
LIN {X 0,Y 255.114,Z 287.528,A -85,B 0,C 180,E1 -19762.052,E2 -19762.052} C_VEL
LIN {X 0,Y 256.172,Z 274.885,A -85,B 0,C 180,E1 -19762.672,E2 -19762.672} C_VEL
LIN {X 0,Y 259.028,Z 214.608,A -85,B 0,C 180,E1 -19764.376,E2 -19764.376} C_VEL
LIN {X 0,Y 253.323,Z 201.5,A -85,B 0,C 180,E1 -19765.836,E2 -19765.836} C_VEL
LIN {X 0,Y 247.27,Z 189.62,A -85,B 0,C 180,E1 -19767.42,E2 -19767.42} C_VEL
LIN {X 0,Y 242.298,Z 181.206,A -85,B 0,C 180,E1 -19768.772,E2 -19768.772} C_VEL
LIN {X 0,Y 239.402,Z 176.905,A -85,B 0,C 180,E1 -19769.578,E2 -19769.578} C_VEL
LIN {X 0,Y 237.419,Z 173.734,A -85,B 0,C 180,E1 -19770.157,E2 -19770.157} C_VEL
LIN {X 0,Y 235.616,Z 171.392,A -85,B 0,C 180,E1 -19770.676,E2 -19770.676} C_VEL
LIN {X 0,Y 234.947,Z 169.217,A -85,B 0,C 180,E1 -19770.962,E2 -19770.962} C_VEL
LIN {X 0,Y 234.985,Z 169.213,A -85,B 0,C 180,E1 -19775.248,E2 -19775.248} C_VEL
LIN {X 0,Y 235.008,Z 169.206,A -85,B 0,C 180,E1 -19778.971,E2 -19778.971} C_VEL
LIN {X 0,Y 235.087,Z 169.194,A -85,B 0,C 180,E1 -19783.068,E2 -19783.068} C_VEL
LIN {X 0,Y 235.109,Z 169.194,A -85,B 0,C 180,E1 -19787.923,E2 -19787.923} C_VEL
LIN {X 0,Y 235.319,Z 169.159,A -85,B 0,C 180,E1 -19791.413,E2 -19791.413} C_VEL
LIN {X 0,Y 235.357,Z 169.167,A -85,B 0,C 180,E1 -19793.141,E2 -19793.141} C_VEL
LIN {X 0,Y 235.593,Z 169.135,A -85,B 0,C 180,E1 -19798.292,E2 -19798.292} C_VEL
LIN {X 0,Y 235.581,Z 169.124,A -85,B 0,C 180,E1 -19801.711,E2 -19801.711} C_VEL
LIN {X 0,Y 235.355,Z 169.152,A -85,B 0,C 180,E1 -19806.861,E2 -19806.861} C_VEL
LIN {X 0,Y 235.213,Z 169.169,A -85,B 0,C 180,E1 -19810.329,E2 -19810.329} C_VEL
LIN {X 0,Y 235.069,Z 169.19,A -85,B 0,C 180,E1 -19815.611,E2 -19815.611} C_VEL
LIN {X 0,Y 235.038,Z 169.194,A -85,B 0,C 180,E1 -19817.091,E2 -19817.091} C_VEL
LIN {X 0,Y 234.273,Z 169.303,A -85,B 0,C 180,E1 -19818.521,E2 -19818.521} C_VEL
LIN {X 0,Y 231.35,Z 169.667,A -85,B 0,C 180,E1 -19820.854,E2 -19820.854} C_VEL
LIN {X 0,Y 228.931,Z 169.966,A -85,B 0,C 180,E1 -19822.756,E2 -19822.756} C_VEL
LIN {X 0,Y 227.914,Z 170.094,A -85,B 0,C 180,E1 -19824.233,E2 -19824.233} C_VEL
LIN {X 0,Y 227.839,Z 170.094,A -85,B 0,C 180,E1 -19824.733,E2 -19824.733} C_VEL
LIN {X 0,Y 227.848,Z 170.097,A -85,B 0,C 180,E1 -19827.561,E2 -19827.561} C_VEL
LIN {X 0,Y 227.858,Z 170.095,A -85,B 0,C 180,E1 -19831.626,E2 -19831.626} C_VEL
LIN {X 0,Y 227.864,Z 170.099,A -85,B 0,C 180,E1 -19835.876,E2 -19835.876} C_VEL
LIN {X 0,Y 227.8,Z 170.109,A -85,B 0,C 180,E1 -19840.384,E2 -19840.384} C_VEL
LIN {X 0,Y 227.852,Z 170.19,A -85,B 0,C 180,E1 -19844.227,E2 -19844.227} C_VEL
LIN {X 0,Y 229.99,Z 177.612,A -85,B 0,C 180,E1 -19848.476,E2 -19848.476} C_VEL
LIN {X 0,Y 230.975,Z 180.872,A -85,B 0,C 180,E1 -19850.143,E2 -19850.143} C_VEL
LIN {X 0,Y 233.47,Z 185.222,A -85,B 0,C 180,E1 -19850.947,E2 -19850.947} C_VEL
LIN {X 0,Y 239.474,Z 195.964,A -85,B 0,C 180,E1 -19852.757,E2 -19852.757} C_VEL
LIN {X 0,Y 245.758,Z 209.077,A -85,B 0,C 180,E1 -19854.569,E2 -19854.569} C_VEL
LIN {X 0,Y 249.815,Z 218.936,A -85,B 0,C 180,E1 -19855.706,E2 -19855.706} C_VEL
LIN {X 0,Y 252.297,Z 238.754,A -85,B 0,C 180,E1 -19856.882,E2 -19856.882} C_VEL
LIN {X 0,Y 249.875,Z 290.642,A -85,B 0,C 180,E1 -19858.422,E2 -19858.422} C_VEL
LIN {X 0,Y 248.407,Z 304.335,A -85,B 0,C 180,E1 -19859.108,E2 -19859.108} C_VEL
LIN {X 0,Y 246.41,Z 317.072,A -85,B 0,C 180,E1 -19860.058,E2 -19860.058} C_VEL
LIN {X 0,Y 244.21,Z 328.08,A -85,B 0,C 180,E1 -19861.181,E2 -19861.181} C_VEL
LIN {X 0,Y 241.574,Z 339.597,A -85,B 0,C 180,E1 -19862.729,E2 -19862.729} C_VEL
LIN {X 0,Y 238.776,Z 350.008,A -85,B 0,C 180,E1 -19864.503,E2 -19864.503} C_VEL
LIN {X 0,Y 236.215,Z 358.546,A -85,B 0,C 180,E1 -19866.318,E2 -19866.318} C_VEL
LIN {X 0,Y 233.863,Z 366.441,A -85,B 0,C 180,E1 -19868.4,E2 -19868.4} C_VEL
LIN {X 0,Y 231.435,Z 374.188,A -85,B 0,C 180,E1 -19870.947,E2 -19870.947} C_VEL
LIN {X 0,Y 229.061,Z 381.346,A -85,B 0,C 180,E1 -19873.971,E2 -19873.971} C_VEL
LIN {X 0,Y 227.484,Z 386.141,A -85,B 0,C 180,E1 -19876.603,E2 -19876.603} C_VEL
LIN {X 0,Y 226.532,Z 389.836,A -85,B 0,C 180,E1 -19879.272,E2 -19879.272} C_VEL
LIN {X 0,Y 226.058,Z 391.762,A -85,B 0,C 180,E1 -19881.058,E2 -19881.058} C_VEL
LIN {X 0,Y 225.773,Z 393.234,A -85,B 0,C 180,E1 -19882.848,E2 -19882.848} C_VEL
LIN {X 0,Y 225.605,Z 394.681,A -85,B 0,C 180,E1 -19885.47,E2 -19885.47} C_VEL
LIN {X 0,Y 225.704,Z 395.254,A -85,B 0,C 180,E1 -19888.216,E2 -19888.216} C_VEL
LIN {X 0,Y 225.82,Z 395.112,A -85,B 0,C 180,E1 -19890,E2 -19890} C_VEL
LIN {X 0,Y 225.728,Z 394.545,A -85,B 0,C 180,E1 -19891.785,E2 -19891.785} C_VEL
LIN {X 0,Y 225.612,Z 392.872,A -85,B 0,C 180,E1 -19894.551,E2 -19894.551} C_VEL
LIN {X 0,Y 225.912,Z 389.296,A -85,B 0,C 180,E1 -19898.048,E2 -19898.048} C_VEL
LIN {X 0,Y 226.476,Z 385.326,A -85,B 0,C 180,E1 -19900.731,E2 -19900.731} C_VEL
LIN {X 0,Y 227.545,Z 379.19,A -85,B 0,C 180,E1 -19903.85,E2 -19903.85} C_VEL
LIN {X 0,Y 229.077,Z 372.472,A -85,B 0,C 180,E1 -19906.487,E2 -19906.487} C_VEL
LIN {X 0,Y 230.827,Z 364.706,A -85,B 0,C 180,E1 -19908.925,E2 -19908.925} C_VEL
LIN {X 0,Y 232.718,Z 355.508,A -85,B 0,C 180,E1 -19911.248,E2 -19911.248} C_VEL
LIN {X 0,Y 235.034,Z 344.896,A -85,B 0,C 180,E1 -19913.342,E2 -19913.342} C_VEL
LIN {X 0,Y 237.081,Z 334.381,A -85,B 0,C 180,E1 -19914.988,E2 -19914.988} C_VEL
LIN {X 0,Y 239.071,Z 322.806,A -85,B 0,C 180,E1 -19916.4,E2 -19916.4} C_VEL
LIN {X 0,Y 240.796,Z 310.826,A -85,B 0,C 180,E1 -19917.485,E2 -19917.485} C_VEL
LIN {X 0,Y 242.116,Z 297.914,A -85,B 0,C 180,E1 -19918.322,E2 -19918.322} C_VEL
LIN {X 0,Y 242.945,Z 284.318,A -85,B 0,C 180,E1 -19918.865,E2 -19918.865} C_VEL
LIN {X 0,Y 244.668,Z 235.772,A -85,B 0,C 180,E1 -19920.298,E2 -19920.298} C_VEL
LIN {X 0,Y 240.649,Z 207.036,A -85,B 0,C 180,E1 -19921.763,E2 -19921.763} C_VEL
LIN {X 0,Y 233.681,Z 189.495,A -85,B 0,C 180,E1 -19923.294,E2 -19923.294} C_VEL
LIN {X 0,Y 230.796,Z 182.524,A -85,B 0,C 180,E1 -19923.961,E2 -19923.961} C_VEL
LIN {X 0,Y 229.131,Z 175.166,A -85,B 0,C 180,E1 -19927.108,E2 -19927.108} C_VEL
LIN {X 0,Y 227.851,Z 170.1,A -85,B 0,C 180,E1 -19929.388,E2 -19929.388} C_VEL
LIN {X 0,Y 227.784,Z 170.102,A -85,B 0,C 180,E1 -19932.749,E2 -19932.749} C_VEL
LIN {X 0,Y 227.814,Z 170.109,A -85,B 0,C 180,E1 -19935.199,E2 -19935.199} C_VEL
LIN {X 0,Y 227.805,Z 170.111,A -85,B 0,C 180,E1 -19939.617,E2 -19939.617} C_VEL
LIN {X 0,Y 227.871,Z 170.101,A -85,B 0,C 180,E1 -19944.125,E2 -19944.125} C_VEL
LIN {X 0,Y 227.861,Z 170.102,A -85,B 0,C 180,E1 -19948.375,E2 -19948.375} C_VEL
LIN {X 0,Y 227.86,Z 170.103,A -85,B 0,C 180,E1 -19952.44,E2 -19952.44} C_VEL
LIN {X 0,Y 227.895,Z 170.098,A -85,B 0,C 180,E1 -19956.364,E2 -19956.364} C_VEL
LIN {X 0,Y 227.895,Z 170.096,A -85,B 0,C 180,E1 -19960.169,E2 -19960.169} C_VEL
LIN {X 0,Y 228.014,Z 170.082,A -85,B 0,C 180,E1 -19963.893,E2 -19963.893} C_VEL
LIN {X 0,Y 228.145,Z 170.059,A -85,B 0,C 180,E1 -19969.347,E2 -19969.347} C_VEL
LIN {X 0,Y 228.305,Z 170.029,A -85,B 0,C 180,E1 -19972.926,E2 -19972.926} C_VEL
LIN {X 0,Y 228.538,Z 170.018,A -85,B 0,C 180,E1 -19978.236,E2 -19978.236} C_VEL
LIN {X 0,Y 228.537,Z 170.002,A -85,B 0,C 180,E1 -19981.761,E2 -19981.761} C_VEL
LIN {X 0,Y 228.307,Z 170.04,A -85,B 0,C 180,E1 -19987.071,E2 -19987.071} C_VEL
LIN {X 0,Y 228.127,Z 170.066,A -85,B 0,C 180,E1 -19990.651,E2 -19990.651} C_VEL
LIN {X 0,Y 228,Z 170.061,A -85,B 0,C 180,E1 -19996.105,E2 -19996.105} C_VEL
LIN {X 0,Y 227.919,Z 170.096,A -85,B 0,C 180,E1 -20001.716,E2 -20001.716} C_VEL
LIN {X 0,Y 227.9,Z 170.078,A -85,B 0,C 180,E1 -20006.579,E2 -20006.579} C_VEL
LIN {X 0,Y 227.868,Z 170.095,A -85,B 0,C 180,E1 -20010.277,E2 -20010.277} C_VEL
LIN {X 0,Y 227.874,Z 170.099,A -85,B 0,C 180,E1 -20013.719,E2 -20013.719} C_VEL
LIN {X 0,Y 227.835,Z 170.086,A -85,B 0,C 180,E1 -20018.091,E2 -20018.091} C_VEL
LIN {X 0,Y 227.783,Z 170.112,A -85,B 0,C 180,E1 -20022.747,E2 -20022.747} C_VEL
LIN {X 0,Y 227.782,Z 170.099,A -85,B 0,C 180,E1 -20027.25,E2 -20027.25} C_VEL
LIN {X 0,Y 227.836,Z 170.106,A -85,B 0,C 180,E1 -20031.907,E2 -20031.907} C_VEL
LIN {X 0,Y 227.874,Z 170.096,A -85,B 0,C 180,E1 -20036.376,E2 -20036.376} C_VEL
LIN {X 0,Y 227.871,Z 170.096,A -85,B 0,C 180,E1 -20040.43,E2 -20040.43} C_VEL
LIN {X 0,Y 227.866,Z 170.102,A -85,B 0,C 180,E1 -20044.418,E2 -20044.418} C_VEL
LIN {X 0,Y 227.913,Z 170.091,A -85,B 0,C 180,E1 -20048.282,E2 -20048.282} C_VEL
LIN {X 0,Y 228.003,Z 170.084,A -85,B 0,C 180,E1 -20053.893,E2 -20053.893} C_VEL
LIN {X 0,Y 228.028,Z 170.083,A -85,B 0,C 180,E1 -20057.778,E2 -20057.778} C_VEL
LIN {X 0,Y 229.238,Z 173.214,A -85,B 0,C 180,E1 -20058.085,E2 -20058.085} C_VEL
LIN {X 0,Y 235.895,Z 185.457,A -85,B 0,C 180,E1 -20059.463,E2 -20059.463} C_VEL
LIN {X 0,Y 245.073,Z 208.291,A -85,B 0,C 180,E1 -20061.42,E2 -20061.42} C_VEL
LIN {X 0,Y 245.565,Z 209.713,A -85,B 0,C 180,E1 -20061.527,E2 -20061.527} C_VEL
LIN {X 0,Y 242.961,Z 274.967,A -85,B 0,C 180,E1 -20063.46,E2 -20063.46} C_VEL
LIN {X 0,Y 241.915,Z 288.256,A -85,B 0,C 180,E1 -20064.164,E2 -20064.164} C_VEL
LIN {X 0,Y 240.556,Z 301.421,A -85,B 0,C 180,E1 -20065.222,E2 -20065.222} C_VEL
LIN {X 0,Y 238.999,Z 312.965,A -85,B 0,C 180,E1 -20066.498,E2 -20066.498} C_VEL
LIN {X 0,Y 237.051,Z 324.187,A -85,B 0,C 180,E1 -20068.088,E2 -20068.088} C_VEL
LIN {X 0,Y 234.97,Z 334.824,A -85,B 0,C 180,E1 -20070,E2 -20070} C_VEL
LIN {X 0,Y 232.781,Z 345.091,A -85,B 0,C 180,E1 -20072.361,E2 -20072.361} C_VEL
LIN {X 0,Y 230.82,Z 353.547,A -85,B 0,C 180,E1 -20074.803,E2 -20074.803} C_VEL
LIN {X 0,Y 229.075,Z 360.933,A -85,B 0,C 180,E1 -20077.492,E2 -20077.492} C_VEL
LIN {X 0,Y 227.846,Z 366.373,A -85,B 0,C 180,E1 -20080.001,E2 -20080.001} C_VEL
LIN {X 0,Y 226.871,Z 370.706,A -85,B 0,C 180,E1 -20082.524,E2 -20082.524} C_VEL
LIN {X 0,Y 226.064,Z 374.496,A -85,B 0,C 180,E1 -20085.482,E2 -20085.482} C_VEL
LIN {X 0,Y 225.612,Z 376.876,A -85,B 0,C 180,E1 -20088.15,E2 -20088.15} C_VEL
LIN {X 0,Y 225.436,Z 378.294,A -85,B 0,C 180,E1 -20090.735,E2 -20090.735} C_VEL
LIN {X 0,Y 225.488,Z 378.878,A -85,B 0,C 180,E1 -20093.902,E2 -20093.902} C_VEL
LIN {X 0,Y 225.692,Z 378.611,A -85,B 0,C 180,E1 -20095.846,E2 -20095.846} C_VEL
LIN {X 0,Y 226.028,Z 377.902,A -85,B 0,C 180,E1 -20097.801,E2 -20097.801} C_VEL
LIN {X 0,Y 226.555,Z 376.682,A -85,B 0,C 180,E1 -20099.758,E2 -20099.758} C_VEL
LIN {X 0,Y 227.572,Z 373.902,A -85,B 0,C 180,E1 -20102.702,E2 -20102.702} C_VEL
LIN {X 0,Y 229.079,Z 369.846,A -85,B 0,C 180,E1 -20105.655,E2 -20105.655} C_VEL
LIN {X 0,Y 231.008,Z 364.401,A -85,B 0,C 180,E1 -20108.585,E2 -20108.585} C_VEL
LIN {X 0,Y 233.473,Z 357.288,A -85,B 0,C 180,E1 -20111.471,E2 -20111.471} C_VEL
LIN {X 0,Y 236.273,Z 348.822,A -85,B 0,C 180,E1 -20114.12,E2 -20114.12} C_VEL
LIN {X 0,Y 239.053,Z 339.623,A -85,B 0,C 180,E1 -20116.382,E2 -20116.382} C_VEL
LIN {X 0,Y 241.711,Z 329.671,A -85,B 0,C 180,E1 -20118.315,E2 -20118.315} C_VEL
LIN {X 0,Y 244.303,Z 318.751,A -85,B 0,C 180,E1 -20119.99,E2 -20119.99} C_VEL
LIN {X 0,Y 246.414,Z 308.135,A -85,B 0,C 180,E1 -20121.271,E2 -20121.271} C_VEL
LIN {X 0,Y 248.361,Z 295.717,A -85,B 0,C 180,E1 -20122.404,E2 -20122.404} C_VEL
LIN {X 0,Y 249.77,Z 282.414,A -85,B 0,C 180,E1 -20123.273,E2 -20123.273} C_VEL
LIN {X 0,Y 250.748,Z 269.96,A -85,B 0,C 180,E1 -20123.756,E2 -20123.756} C_VEL
LIN {X 0,Y 253.18,Z 216.294,A -85,B 0,C 180,E1 -20125.313,E2 -20125.313} C_VEL
LIN {X 0,Y 247.73,Z 203.965,A -85,B 0,C 180,E1 -20126.771,E2 -20126.771} C_VEL
LIN {X 0,Y 241.864,Z 192.521,A -85,B 0,C 180,E1 -20128.4,E2 -20128.4} C_VEL
LIN {X 0,Y 238.002,Z 186.002,A -85,B 0,C 180,E1 -20129.502,E2 -20129.502} C_VEL
LIN {X 0,Y 233.173,Z 178.707,A -85,B 0,C 180,E1 -20130.936,E2 -20130.936} C_VEL
LIN {X 0,Y 230.594,Z 174.847,A -85,B 0,C 180,E1 -20131.749,E2 -20131.749} C_VEL
LIN {X 0,Y 228.642,Z 172.534,A -85,B 0,C 180,E1 -20132.359,E2 -20132.359} C_VEL
LIN {X 0,Y 227.899,Z 170.095,A -85,B 0,C 180,E1 -20132.682,E2 -20132.682} C_VEL
LIN {X 0,Y 227.912,Z 170.093,A -85,B 0,C 180,E1 -20136.369,E2 -20136.369} C_VEL
LIN {X 0,Y 227.936,Z 170.092,A -85,B 0,C 180,E1 -20140.176,E2 -20140.176} C_VEL
LIN {X 0,Y 228.042,Z 170.076,A -85,B 0,C 180,E1 -20143.898,E2 -20143.898} C_VEL
LIN {X 0,Y 228.066,Z 170.068,A -85,B 0,C 180,E1 -20147.544,E2 -20147.544} C_VEL
LIN {X 0,Y 228.258,Z 170.038,A -85,B 0,C 180,E1 -20151.146,E2 -20151.146} C_VEL
LIN {X 0,Y 228.309,Z 170.042,A -85,B 0,C 180,E1 -20152.929,E2 -20152.929} C_VEL
LIN {X 0,Y 228.551,Z 170.012,A -85,B 0,C 180,E1 -20158.239,E2 -20158.239} C_VEL
LIN {X 0,Y 228.539,Z 170.001,A -85,B 0,C 180,E1 -20161.764,E2 -20161.764} C_VEL
LIN {X 0,Y 228.308,Z 170.032,A -85,B 0,C 180,E1 -20167.074,E2 -20167.074} C_VEL
LIN {X 0,Y 228.143,Z 170.047,A -85,B 0,C 180,E1 -20170.653,E2 -20170.653} C_VEL
LIN {X 0,Y 228.03,Z 170.079,A -85,B 0,C 180,E1 -20174.276,E2 -20174.276} C_VEL
LIN {X 0,Y 227.93,Z 170.087,A -85,B 0,C 180,E1 -20177.961,E2 -20177.961} C_VEL
LIN {X 0,Y 227.893,Z 170.086,A -85,B 0,C 180,E1 -20182.306,E2 -20182.306} C_VEL
LIN {X 0,Y 227.839,Z 170.094,A -85,B 0,C 180,E1 -20184.733,E2 -20184.733} C_VEL
LIN {X 0,Y 227.177,Z 170.177,A -85,B 0,C 180,E1 -20186.208,E2 -20186.208} C_VEL
LIN {X 0,Y 224.292,Z 170.547,A -85,B 0,C 180,E1 -20188.613,E2 -20188.613} C_VEL
LIN {X 0,Y 221.861,Z 170.842,A -85,B 0,C 180,E1 -20190.576,E2 -20190.576} C_VEL
LIN {X 0,Y 220.863,Z 170.971,A -85,B 0,C 180,E1 -20192.102,E2 -20192.102} C_VEL
LIN {X 0,Y 220.806,Z 170.98,A -85,B 0,C 180,E1 -20192.618,E2 -20192.618} C_VEL
LIN {X 0,Y 220.799,Z 170.976,A -85,B 0,C 180,E1 -20197.274,E2 -20197.274} C_VEL
LIN {X 0,Y 220.748,Z 170.987,A -85,B 0,C 180,E1 -20201.959,E2 -20201.959} C_VEL
LIN {X 0,Y 220.765,Z 171.169,A -85,B 0,C 180,E1 -20202.621,E2 -20202.621} C_VEL
LIN {X 0,Y 222.691,Z 177.45,A -85,B 0,C 180,E1 -20206.543,E2 -20206.543} C_VEL
LIN {X 0,Y 223.589,Z 180.511,A -85,B 0,C 180,E1 -20208.185,E2 -20208.185} C_VEL
LIN {X 0,Y 226.078,Z 184.729,A -85,B 0,C 180,E1 -20209.064,E2 -20209.064} C_VEL
LIN {X 0,Y 227.638,Z 187.263,A -85,B 0,C 180,E1 -20209.593,E2 -20209.593} C_VEL
LIN {X 0,Y 230.678,Z 192.423,A -85,B 0,C 180,E1 -20210.595,E2 -20210.595} C_VEL
LIN {X 0,Y 236.844,Z 204.069,A -85,B 0,C 180,E1 -20212.526,E2 -20212.526} C_VEL
LIN {X 0,Y 243.098,Z 218.133,A -85,B 0,C 180,E1 -20214.406,E2 -20214.406} C_VEL
LIN {X 0,Y 244.51,Z 222.171,A -85,B 0,C 180,E1 -20214.841,E2 -20214.841} C_VEL
LIN {X 0,Y 246.632,Z 240.014,A -85,B 0,C 180,E1 -20215.925,E2 -20215.925} C_VEL
LIN {X 0,Y 244.098,Z 290.912,A -85,B 0,C 180,E1 -20217.467,E2 -20217.467} C_VEL
LIN {X 0,Y 242.522,Z 304.959,A -85,B 0,C 180,E1 -20218.198,E2 -20218.198} C_VEL
LIN {X 0,Y 240.505,Z 317.017,A -85,B 0,C 180,E1 -20219.122,E2 -20219.122} C_VEL
LIN {X 0,Y 238.045,Z 328.747,A -85,B 0,C 180,E1 -20220.362,E2 -20220.362} C_VEL
LIN {X 0,Y 235.315,Z 340.074,A -85,B 0,C 180,E1 -20221.94,E2 -20221.94} C_VEL
LIN {X 0,Y 232.417,Z 350.339,A -85,B 0,C 180,E1 -20223.753,E2 -20223.753} C_VEL
LIN {X 0,Y 229.728,Z 358.764,A -85,B 0,C 180,E1 -20225.607,E2 -20225.607} C_VEL
LIN {X 0,Y 226.822,Z 367.929,A -85,B 0,C 180,E1 -20228.173,E2 -20228.173} C_VEL
LIN {X 0,Y 224.314,Z 375.347,A -85,B 0,C 180,E1 -20230.794,E2 -20230.794} C_VEL
LIN {X 0,Y 222.24,Z 381.326,A -85,B 0,C 180,E1 -20233.465,E2 -20233.465} C_VEL
LIN {X 0,Y 220.554,Z 386.07,A -85,B 0,C 180,E1 -20236.173,E2 -20236.173} C_VEL
LIN {X 0,Y 219.53,Z 389.717,A -85,B 0,C 180,E1 -20238.926,E2 -20238.926} C_VEL
LIN {X 0,Y 219.022,Z 391.612,A -85,B 0,C 180,E1 -20240.768,E2 -20240.768} C_VEL
LIN {X 0,Y 218.568,Z 394.086,A -85,B 0,C 180,E1 -20244.465,E2 -20244.465} C_VEL
LIN {X 0,Y 218.617,Z 394.999,A -85,B 0,C 180,E1 -20248.158,E2 -20248.158} C_VEL
LIN {X 0,Y 218.729,Z 394.822,A -85,B 0,C 180,E1 -20250,E2 -20250} C_VEL
LIN {X 0,Y 218.639,Z 394.236,A -85,B 0,C 180,E1 -20251.842,E2 -20251.842} C_VEL
LIN {X 0,Y 218.524,Z 392.738,A -85,B 0,C 180,E1 -20254.426,E2 -20254.426} C_VEL
LIN {X 0,Y 218.751,Z 389.982,A -85,B 0,C 180,E1 -20257.384,E2 -20257.384} C_VEL
LIN {X 0,Y 219.224,Z 386.33,A -85,B 0,C 180,E1 -20260.156,E2 -20260.156} C_VEL
LIN {X 0,Y 220.011,Z 381.537,A -85,B 0,C 180,E1 -20262.921,E2 -20262.921} C_VEL
LIN {X 0,Y 221.706,Z 374.349,A -85,B 0,C 180,E1 -20266.104,E2 -20266.104} C_VEL
LIN {X 0,Y 223.495,Z 366.749,A -85,B 0,C 180,E1 -20268.72,E2 -20268.72} C_VEL
LIN {X 0,Y 225.274,Z 358.418,A -85,B 0,C 180,E1 -20271.025,E2 -20271.025} C_VEL
LIN {X 0,Y 227.466,Z 348.59,A -85,B 0,C 180,E1 -20273.2,E2 -20273.2} C_VEL
LIN {X 0,Y 229.793,Z 337.661,A -85,B 0,C 180,E1 -20275.11,E2 -20275.11} C_VEL
LIN {X 0,Y 231.822,Z 326.97,A -85,B 0,C 180,E1 -20276.563,E2 -20276.563} C_VEL
LIN {X 0,Y 233.817,Z 314.118,A -85,B 0,C 180,E1 -20277.89,E2 -20277.89} C_VEL
LIN {X 0,Y 235.366,Z 301.167,A -85,B 0,C 180,E1 -20278.844,E2 -20278.844} C_VEL
LIN {X 0,Y 236.324,Z 288.452,A -85,B 0,C 180,E1 -20279.448,E2 -20279.448} C_VEL
LIN {X 0,Y 238.296,Z 236.307,A -85,B 0,C 180,E1 -20281.038,E2 -20281.038} C_VEL
LIN {X 0,Y 234.544,Z 209.248,A -85,B 0,C 180,E1 -20282.466,E2 -20282.466} C_VEL
LIN {X 0,Y 227.662,Z 192.003,A -85,B 0,C 180,E1 -20284.046,E2 -20284.046} C_VEL
LIN {X 0,Y 223.505,Z 182.229,A -85,B 0,C 180,E1 -20285.041,E2 -20285.041} C_VEL
LIN {X 0,Y 221.558,Z 173.989,A -85,B 0,C 180,E1 -20288.748,E2 -20288.748} C_VEL
LIN {X 0,Y 220.773,Z 170.988,A -85,B 0,C 180,E1 -20290.179,E2 -20290.179} C_VEL
LIN {X 0,Y 220.756,Z 170.987,A -85,B 0,C 180,E1 -20294.459,E2 -20294.459} C_VEL
LIN {X 0,Y 220.753,Z 170.988,A -85,B 0,C 180,E1 -20298.042,E2 -20298.042} C_VEL
LIN {X 0,Y 220.83,Z 170.98,A -85,B 0,C 180,E1 -20302.792,E2 -20302.792} C_VEL
LIN {X 0,Y 220.817,Z 170.982,A -85,B 0,C 180,E1 -20307.242,E2 -20307.242} C_VEL
LIN {X 0,Y 220.809,Z 170.981,A -85,B 0,C 180,E1 -20311.481,E2 -20311.481} C_VEL
LIN {X 0,Y 220.85,Z 170.974,A -85,B 0,C 180,E1 -20315.561,E2 -20315.561} C_VEL
LIN {X 0,Y 220.854,Z 170.972,A -85,B 0,C 180,E1 -20319.509,E2 -20319.509} C_VEL
LIN {X 0,Y 220.974,Z 170.958,A -85,B 0,C 180,E1 -20323.365,E2 -20323.365} C_VEL
LIN {X 0,Y 221.064,Z 170.941,A -85,B 0,C 180,E1 -20329.002,E2 -20329.002} C_VEL
LIN {X 0,Y 221.242,Z 170.906,A -85,B 0,C 180,E1 -20332.699,E2 -20332.699} C_VEL
LIN {X 0,Y 221.472,Z 170.899,A -85,B 0,C 180,E1 -20338.18,E2 -20338.18} C_VEL
LIN {X 0,Y 221.47,Z 170.88,A -85,B 0,C 180,E1 -20341.817,E2 -20341.817} C_VEL
LIN {X 0,Y 221.244,Z 170.92,A -85,B 0,C 180,E1 -20347.298,E2 -20347.298} C_VEL
LIN {X 0,Y 221.051,Z 170.947,A -85,B 0,C 180,E1 -20350.996,E2 -20350.996} C_VEL
LIN {X 0,Y 220.967,Z 170.939,A -85,B 0,C 180,E1 -20356.632,E2 -20356.632} C_VEL
LIN {X 0,Y 220.846,Z 170.973,A -85,B 0,C 180,E1 -20360.489,E2 -20360.489} C_VEL
LIN {X 0,Y 220.796,Z 170.974,A -85,B 0,C 180,E1 -20364.442,E2 -20364.442} C_VEL
LIN {X 0,Y 220.794,Z 170.964,A -85,B 0,C 180,E1 -20368.518,E2 -20368.518} C_VEL
LIN {X 0,Y 220.81,Z 170.979,A -85,B 0,C 180,E1 -20372.755,E2 -20372.755} C_VEL
LIN {X 0,Y 220.794,Z 170.964,A -85,B 0,C 180,E1 -20377.271,E2 -20377.271} C_VEL
LIN {X 0,Y 220.746,Z 170.988,A -85,B 0,C 180,E1 -20381.956,E2 -20381.956} C_VEL
LIN {X 0,Y 220.75,Z 170.98,A -85,B 0,C 180,E1 -20385.539,E2 -20385.539} C_VEL
LIN {X 0,Y 220.777,Z 170.985,A -85,B 0,C 180,E1 -20390.456,E2 -20390.456} C_VEL
LIN {X 0,Y 220.821,Z 170.979,A -85,B 0,C 180,E1 -20392.791,E2 -20392.791} C_VEL
LIN {X 0,Y 220.808,Z 170.983,A -85,B 0,C 180,E1 -20397.242,E2 -20397.242} C_VEL
LIN {X 0,Y 220.794,Z 170.974,A -85,B 0,C 180,E1 -20401.48,E2 -20401.48} C_VEL
LIN {X 0,Y 220.797,Z 170.976,A -85,B 0,C 180,E1 -20405.556,E2 -20405.556} C_VEL
LIN {X 0,Y 220.84,Z 170.977,A -85,B 0,C 180,E1 -20409.508,E2 -20409.508} C_VEL
LIN {X 0,Y 220.964,Z 170.96,A -85,B 0,C 180,E1 -20413.366,E2 -20413.366} C_VEL
LIN {X 0,Y 220.949,Z 170.959,A -85,B 0,C 180,E1 -20416.725,E2 -20416.725} C_VEL
LIN {X 0,Y 221.951,Z 173.799,A -85,B 0,C 180,E1 -20417.016,E2 -20417.016} C_VEL
LIN {X 0,Y 225.116,Z 179.293,A -85,B 0,C 180,E1 -20417.708,E2 -20417.708} C_VEL
LIN {X 0,Y 231.078,Z 190.622,A -85,B 0,C 180,E1 -20418.989,E2 -20418.989} C_VEL
LIN {X 0,Y 239.275,Z 211.512,A -85,B 0,C 180,E1 -20420.821,E2 -20420.821} C_VEL
LIN {X 0,Y 236.522,Z 275.529,A -85,B 0,C 180,E1 -20422.756,E2 -20422.756} C_VEL
LIN {X 0,Y 235.457,Z 288.548,A -85,B 0,C 180,E1 -20423.465,E2 -20423.465} C_VEL
LIN {X 0,Y 234.093,Z 301.281,A -85,B 0,C 180,E1 -20424.508,E2 -20424.508} C_VEL
LIN {X 0,Y 232.546,Z 312.685,A -85,B 0,C 180,E1 -20425.785,E2 -20425.785} C_VEL
LIN {X 0,Y 230.533,Z 323.804,A -85,B 0,C 180,E1 -20427.379,E2 -20427.379} C_VEL
LIN {X 0,Y 228.369,Z 334.55,A -85,B 0,C 180,E1 -20429.338,E2 -20429.338} C_VEL
LIN {X 0,Y 226.473,Z 343.302,A -85,B 0,C 180,E1 -20431.333,E2 -20431.333} C_VEL
LIN {X 0,Y 224.184,Z 352.771,A -85,B 0,C 180,E1 -20434.044,E2 -20434.044} C_VEL
LIN {X 0,Y 222.332,Z 360.359,A -85,B 0,C 180,E1 -20436.807,E2 -20436.807} C_VEL
LIN {X 0,Y 220.921,Z 366.281,A -85,B 0,C 180,E1 -20439.547,E2 -20439.547} C_VEL
LIN {X 0,Y 219.944,Z 370.428,A -85,B 0,C 180,E1 -20441.987,E2 -20441.987} C_VEL
LIN {X 0,Y 219.111,Z 374.201,A -85,B 0,C 180,E1 -20444.868,E2 -20444.868} C_VEL
LIN {X 0,Y 218.709,Z 376.099,A -85,B 0,C 180,E1 -20446.81,E2 -20446.81} C_VEL
LIN {X 0,Y 218.444,Z 377.524,A -85,B 0,C 180,E1 -20448.767,E2 -20448.767} C_VEL
LIN {X 0,Y 218.338,Z 378.628,A -85,B 0,C 180,E1 -20451.023,E2 -20451.023} C_VEL
LIN {X 0,Y 218.478,Z 379.096,A -85,B 0,C 180,E1 -20454.72,E2 -20454.72} C_VEL
LIN {X 0,Y 218.717,Z 378.72,A -85,B 0,C 180,E1 -20456.734,E2 -20456.734} C_VEL
LIN {X 0,Y 219.575,Z 376.884,A -85,B 0,C 180,E1 -20460.213,E2 -20460.213} C_VEL
LIN {X 0,Y 220.498,Z 374.575,A -85,B 0,C 180,E1 -20462.809,E2 -20462.809} C_VEL
LIN {X 0,Y 222.038,Z 370.677,A -85,B 0,C 180,E1 -20465.843,E2 -20465.843} C_VEL
LIN {X 0,Y 224.044,Z 365.392,A -85,B 0,C 180,E1 -20468.857,E2 -20468.857} C_VEL
LIN {X 0,Y 226.669,Z 358.287,A -85,B 0,C 180,E1 -20471.918,E2 -20471.918} C_VEL
LIN {X 0,Y 229.678,Z 349.671,A -85,B 0,C 180,E1 -20474.731,E2 -20474.731} C_VEL
LIN {X 0,Y 232.658,Z 340.416,A -85,B 0,C 180,E1 -20477.099,E2 -20477.099} C_VEL
LIN {X 0,Y 235.504,Z 330.348,A -85,B 0,C 180,E1 -20479.119,E2 -20479.119} C_VEL
LIN {X 0,Y 238.129,Z 319.855,A -85,B 0,C 180,E1 -20480.78,E2 -20480.78} C_VEL
LIN {X 0,Y 240.58,Z 308.083,A -85,B 0,C 180,E1 -20482.239,E2 -20482.239} C_VEL
LIN {X 0,Y 242.553,Z 296.077,A -85,B 0,C 180,E1 -20483.345,E2 -20483.345} C_VEL
LIN {X 0,Y 244.022,Z 282.9,A -85,B 0,C 180,E1 -20484.223,E2 -20484.223} C_VEL
LIN {X 0,Y 245.02,Z 270.551,A -85,B 0,C 180,E1 -20484.719,E2 -20484.719} C_VEL
LIN {X 0,Y 247.503,Z 218.499,A -85,B 0,C 180,E1 -20486.255,E2 -20486.255} C_VEL
LIN {X 0,Y 242.589,Z 207.248,A -85,B 0,C 180,E1 -20487.654,E2 -20487.654} C_VEL
LIN {X 0,Y 237.116,Z 196.513,A -85,B 0,C 180,E1 -20489.253,E2 -20489.253} C_VEL
LIN {X 0,Y 232.298,Z 188.343,A -85,B 0,C 180,E1 -20490.716,E2 -20490.716} C_VEL
LIN {X 0,Y 226.723,Z 180.206,A -85,B 0,C 180,E1 -20492.498,E2 -20492.498} C_VEL
LIN {X 0,Y 224.426,Z 176.925,A -85,B 0,C 180,E1 -20493.276,E2 -20493.276} C_VEL
LIN {X 0,Y 223.677,Z 175.772,A -85,B 0,C 180,E1 -20493.539,E2 -20493.539} C_VEL
LIN {X 0,Y 221.676,Z 173.456,A -85,B 0,C 180,E1 -20494.22,E2 -20494.22} C_VEL
LIN {X 0,Y 220.894,Z 170.972,A -85,B 0,C 180,E1 -20494.628,E2 -20494.628} C_VEL
LIN {X 0,Y 220.895,Z 170.974,A -85,B 0,C 180,E1 -20497.557,E2 -20497.557} C_VEL
LIN {X 0,Y 220.978,Z 170.951,A -85,B 0,C 180,E1 -20502.577,E2 -20502.577} C_VEL
LIN {X 0,Y 221.004,Z 170.945,A -85,B 0,C 180,E1 -20507.14,E2 -20507.14} C_VEL
LIN {X 0,Y 221.197,Z 170.918,A -85,B 0,C 180,E1 -20510.861,E2 -20510.861} C_VEL
LIN {X 0,Y 221.125,Z 170.93,A -85,B 0,C 180,E1 -20514.53,E2 -20514.53} C_VEL
LIN {X 0,Y 221.509,Z 170.889,A -85,B 0,C 180,E1 -20518.183,E2 -20518.183} C_VEL
LIN {X 0,Y 221.472,Z 170.881,A -85,B 0,C 180,E1 -20521.82,E2 -20521.82} C_VEL
LIN {X 0,Y 221.245,Z 170.913,A -85,B 0,C 180,E1 -20527.301,E2 -20527.301} C_VEL
LIN {X 0,Y 221.062,Z 170.928,A -85,B 0,C 180,E1 -20530.998,E2 -20530.998} C_VEL
LIN {X 0,Y 220.977,Z 170.943,A -85,B 0,C 180,E1 -20536.634,E2 -20536.634} C_VEL
LIN {X 0,Y 220.852,Z 170.964,A -85,B 0,C 180,E1 -20540.492,E2 -20540.492} C_VEL
LIN {X 0,Y 220.796,Z 170.977,A -85,B 0,C 180,E1 -20544.724,E2 -20544.724} C_VEL
LIN {X 0,Y 220.802,Z 170.981,A -85,B 0,C 180,E1 -20548.52,E2 -20548.52} C_VEL
LIN {X 0,Y 220.806,Z 170.98,A -85,B 0,C 180,E1 -20552.618,E2 -20552.618} C_VEL
LIN {X 0,Y 220.17,Z 171.068,A -85,B 0,C 180,E1 -20553.631,E2 -20553.631} C_VEL
LIN {X 0,Y 217.34,Z 171.42,A -85,B 0,C 180,E1 -20555.222,E2 -20555.222} C_VEL
LIN {X 0,Y 214.429,Z 171.774,A -85,B 0,C 180,E1 -20556.853,E2 -20556.853} C_VEL
LIN {X 0,Y 213.714,Z 171.857,A -85,B 0,C 180,E1 -20557.912,E2 -20557.912} C_VEL
LIN {X 0,Y 213.71,Z 171.931,A -85,B 0,C 180,E1 -20560.695,E2 -20560.695} C_VEL
LIN {X 0,Y 215.462,Z 177.608,A -85,B 0,C 180,E1 -20564.564,E2 -20564.564} C_VEL
LIN {X 0,Y 216.257,Z 180.127,A -85,B 0,C 180,E1 -20566.022,E2 -20566.022} C_VEL
LIN {X 0,Y 218.951,Z 184.524,A -85,B 0,C 180,E1 -20567.066,E2 -20567.066} C_VEL
LIN {X 0,Y 223.739,Z 192.371,A -85,B 0,C 180,E1 -20568.807,E2 -20568.807} C_VEL
LIN {X 0,Y 226.869,Z 197.824,A -85,B 0,C 180,E1 -20569.891,E2 -20569.891} C_VEL
LIN {X 0,Y 232.441,Z 208.614,A -85,B 0,C 180,E1 -20571.735,E2 -20571.735} C_VEL
LIN {X 0,Y 238.286,Z 222.04,A -85,B 0,C 180,E1 -20573.582,E2 -20573.582} C_VEL
LIN {X 0,Y 239.19,Z 224.401,A -85,B 0,C 180,E1 -20573.867,E2 -20573.867} C_VEL
LIN {X 0,Y 241.053,Z 241.22,A -85,B 0,C 180,E1 -20574.922,E2 -20574.922} C_VEL
LIN {X 0,Y 238.421,Z 290.801,A -85,B 0,C 180,E1 -20576.448,E2 -20576.448} C_VEL
LIN {X 0,Y 236.881,Z 304.195,A -85,B 0,C 180,E1 -20577.154,E2 -20577.154} C_VEL
LIN {X 0,Y 234.682,Z 316.954,A -85,B 0,C 180,E1 -20578.142,E2 -20578.142} C_VEL
LIN {X 0,Y 231.923,Z 329.426,A -85,B 0,C 180,E1 -20579.498,E2 -20579.498} C_VEL
LIN {X 0,Y 229.112,Z 340.581,A -85,B 0,C 180,E1 -20581.11,E2 -20581.11} C_VEL
LIN {X 0,Y 226.083,Z 350.685,A -85,B 0,C 180,E1 -20582.959,E2 -20582.959} C_VEL
LIN {X 0,Y 222.719,Z 360.635,A -85,B 0,C 180,E1 -20585.285,E2 -20585.285} C_VEL
LIN {X 0,Y 219.865,Z 369.133,A -85,B 0,C 180,E1 -20587.833,E2 -20587.833} C_VEL
LIN {X 0,Y 217.623,Z 375.402,A -85,B 0,C 180,E1 -20590.179,E2 -20590.179} C_VEL
LIN {X 0,Y 215.441,Z 381.312,A -85,B 0,C 180,E1 -20592.927,E2 -20592.927} C_VEL
LIN {X 0,Y 213.647,Z 385.999,A -85,B 0,C 180,E1 -20595.717,E2 -20595.717} C_VEL
LIN {X 0,Y 212.521,Z 389.598,A -85,B 0,C 180,E1 -20598.556,E2 -20598.556} C_VEL
LIN {X 0,Y 212.004,Z 391.452,A -85,B 0,C 180,E1 -20600.459,E2 -20600.459} C_VEL
LIN {X 0,Y 211.489,Z 393.879,A -85,B 0,C 180,E1 -20604.279,E2 -20604.279} C_VEL
LIN {X 0,Y 211.441,Z 394.509,A -85,B 0,C 180,E1 -20606.189,E2 -20606.189} C_VEL
LIN {X 0,Y 211.512,Z 394.734,A -85,B 0,C 180,E1 -20608.096,E2 -20608.096} C_VEL
LIN {X 0,Y 211.641,Z 394.529,A -85,B 0,C 180,E1 -20610,E2 -20610} C_VEL
LIN {X 0,Y 211.552,Z 393.921,A -85,B 0,C 180,E1 -20611.904,E2 -20611.904} C_VEL
LIN {X 0,Y 211.427,Z 392.622,A -85,B 0,C 180,E1 -20614.254,E2 -20614.254} C_VEL
LIN {X 0,Y 211.675,Z 389.573,A -85,B 0,C 180,E1 -20617.632,E2 -20617.632} C_VEL
LIN {X 0,Y 212.188,Z 385.871,A -85,B 0,C 180,E1 -20620.497,E2 -20620.497} C_VEL
LIN {X 0,Y 213.051,Z 381.023,A -85,B 0,C 180,E1 -20623.351,E2 -20623.351} C_VEL
LIN {X 0,Y 214.557,Z 374.905,A -85,B 0,C 180,E1 -20626.167,E2 -20626.167} C_VEL
LIN {X 0,Y 216.468,Z 367.277,A -85,B 0,C 180,E1 -20628.946,E2 -20628.946} C_VEL
LIN {X 0,Y 218.216,Z 359.447,A -85,B 0,C 180,E1 -20631.244,E2 -20631.244} C_VEL
LIN {X 0,Y 220.374,Z 349.879,A -85,B 0,C 180,E1 -20633.494,E2 -20633.494} C_VEL
LIN {X 0,Y 222.781,Z 339.288,A -85,B 0,C 180,E1 -20635.457,E2 -20635.457} C_VEL
LIN {X 0,Y 225.143,Z 327.483,A -85,B 0,C 180,E1 -20637.164,E2 -20637.164} C_VEL
LIN {X 0,Y 227.204,Z 314.85,A -85,B 0,C 180,E1 -20638.524,E2 -20638.524} C_VEL
LIN {X 0,Y 228.882,Z 301.654,A -85,B 0,C 180,E1 -20639.544,E2 -20639.544} C_VEL
LIN {X 0,Y 229.896,Z 289.351,A -85,B 0,C 180,E1 -20640.164,E2 -20640.164} C_VEL
LIN {X 0,Y 231.918,Z 236.732,A -85,B 0,C 180,E1 -20641.823,E2 -20641.823} C_VEL
LIN {X 0,Y 228.436,Z 211.508,A -85,B 0,C 180,E1 -20643.21,E2 -20643.21} C_VEL
LIN {X 0,Y 220.909,Z 192.584,A -85,B 0,C 180,E1 -20645.021,E2 -20645.021} C_VEL
LIN {X 0,Y 216.201,Z 181.821,A -85,B 0,C 180,E1 -20646.245,E2 -20646.245} C_VEL
LIN {X 0,Y 214.093,Z 173.38,A -85,B 0,C 180,E1 -20650.249,E2 -20650.249} C_VEL
LIN {X 0,Y 213.711,Z 171.861,A -85,B 0,C 180,E1 -20651.018,E2 -20651.018} C_VEL
LIN {X 0,Y 213.706,Z 171.86,A -85,B 0,C 180,E1 -20653.68,E2 -20653.68} C_VEL
LIN {X 0,Y 213.706,Z 171.865,A -85,B 0,C 180,E1 -20656.345,E2 -20656.345} C_VEL
LIN {X 0,Y 213.709,Z 171.868,A -85,B 0,C 180,E1 -20661.329,E2 -20661.329} C_VEL
LIN {X 0,Y 213.759,Z 171.859,A -85,B 0,C 180,E1 -20666.017,E2 -20666.017} C_VEL
LIN {X 0,Y 213.755,Z 171.86,A -85,B 0,C 180,E1 -20670.449,E2 -20670.449} C_VEL
LIN {X 0,Y 213.786,Z 171.856,A -85,B 0,C 180,E1 -20674.698,E2 -20674.698} C_VEL
LIN {X 0,Y 213.782,Z 171.856,A -85,B 0,C 180,E1 -20678.799,E2 -20678.799} C_VEL
LIN {X 0,Y 213.884,Z 171.843,A -85,B 0,C 180,E1 -20682.797,E2 -20682.797} C_VEL
LIN {X 0,Y 213.921,Z 171.839,A -85,B 0,C 180,E1 -20686.703,E2 -20686.703} C_VEL
LIN {X 0,Y 214.138,Z 171.793,A -85,B 0,C 180,E1 -20690.554,E2 -20690.554} C_VEL
LIN {X 0,Y 214.079,Z 171.807,A -85,B 0,C 180,E1 -20694.346,E2 -20694.346} C_VEL
LIN {X 0,Y 214.409,Z 171.779,A -85,B 0,C 180,E1 -20698.12,E2 -20698.12} C_VEL
LIN {X 0,Y 214.516,Z 171.758,A -85,B 0,C 180,E1 -20699.998,E2 -20699.998} C_VEL
LIN {X 0,Y 214.407,Z 171.758,A -85,B 0,C 180,E1 -20701.877,E2 -20701.877} C_VEL
LIN {X 0,Y 214.185,Z 171.8,A -85,B 0,C 180,E1 -20707.54,E2 -20707.54} C_VEL
LIN {X 0,Y 213.984,Z 171.828,A -85,B 0,C 180,E1 -20711.364,E2 -20711.364} C_VEL
LIN {X 0,Y 213.866,Z 171.819,A -85,B 0,C 180,E1 -20715.24,E2 -20715.24} C_VEL
LIN {X 0,Y 213.791,Z 171.847,A -85,B 0,C 180,E1 -20719.19,E2 -20719.19} C_VEL
LIN {X 0,Y 213.783,Z 171.854,A -85,B 0,C 180,E1 -20723.233,E2 -20723.233} C_VEL
LIN {X 0,Y 213.784,Z 171.831,A -85,B 0,C 180,E1 -20727.425,E2 -20727.425} C_VEL
LIN {X 0,Y 213.757,Z 171.858,A -85,B 0,C 180,E1 -20731.737,E2 -20731.737} C_VEL
LIN {X 0,Y 213.739,Z 171.85,A -85,B 0,C 180,E1 -20736.287,E2 -20736.287} C_VEL
LIN {X 0,Y 213.696,Z 171.863,A -85,B 0,C 180,E1 -20741.127,E2 -20741.127} C_VEL
LIN {X 0,Y 213.698,Z 171.866,A -85,B 0,C 180,E1 -20743.678,E2 -20743.678} C_VEL
LIN {X 0,Y 213.698,Z 171.855,A -85,B 0,C 180,E1 -20746.344,E2 -20746.344} C_VEL
LIN {X 0,Y 213.7,Z 171.869,A -85,B 0,C 180,E1 -20751.328,E2 -20751.328} C_VEL
LIN {X 0,Y 213.75,Z 171.854,A -85,B 0,C 180,E1 -20756.016,E2 -20756.016} C_VEL
LIN {X 0,Y 213.743,Z 171.854,A -85,B 0,C 180,E1 -20760.448,E2 -20760.448} C_VEL
LIN {X 0,Y 213.745,Z 171.858,A -85,B 0,C 180,E1 -20764.694,E2 -20764.694} C_VEL
LIN {X 0,Y 213.769,Z 171.856,A -85,B 0,C 180,E1 -20768.798,E2 -20768.798} C_VEL
LIN {X 0,Y 213.873,Z 171.843,A -85,B 0,C 180,E1 -20772.797,E2 -20772.797} C_VEL
LIN {X 0,Y 213.913,Z 171.921,A -85,B 0,C 180,E1 -20775.637,E2 -20775.637} C_VEL
LIN {X 0,Y 214.948,Z 174.757,A -85,B 0,C 180,E1 -20775.927,E2 -20775.927} C_VEL
LIN {X 0,Y 221.505,Z 186.337,A -85,B 0,C 180,E1 -20777.433,E2 -20777.433} C_VEL
LIN {X 0,Y 226.069,Z 195.414,A -85,B 0,C 180,E1 -20778.456,E2 -20778.456} C_VEL
LIN {X 0,Y 232.868,Z 212.865,A -85,B 0,C 180,E1 -20780.041,E2 -20780.041} C_VEL
LIN {X 0,Y 230.155,Z 275.371,A -85,B 0,C 180,E1 -20781.98,E2 -20781.98} C_VEL
LIN {X 0,Y 229.089,Z 288.391,A -85,B 0,C 180,E1 -20782.699,E2 -20782.699} C_VEL
LIN {X 0,Y 227.607,Z 301.559,A -85,B 0,C 180,E1 -20783.795,E2 -20783.795} C_VEL
LIN {X 0,Y 225.967,Z 313.148,A -85,B 0,C 180,E1 -20785.131,E2 -20785.131} C_VEL
LIN {X 0,Y 223.786,Z 324.731,A -85,B 0,C 180,E1 -20786.849,E2 -20786.849} C_VEL
LIN {X 0,Y 221.564,Z 335.358,A -85,B 0,C 180,E1 -20788.864,E2 -20788.864} C_VEL
LIN {X 0,Y 219.596,Z 344.01,A -85,B 0,C 180,E1 -20790.917,E2 -20790.917} C_VEL
LIN {X 0,Y 217.214,Z 353.389,A -85,B 0,C 180,E1 -20793.71,E2 -20793.71} C_VEL
LIN {X 0,Y 215.322,Z 360.913,A -85,B 0,C 180,E1 -20796.559,E2 -20796.559} C_VEL
LIN {X 0,Y 213.8,Z 367.058,A -85,B 0,C 180,E1 -20799.556,E2 -20799.556} C_VEL
LIN {X 0,Y 212.699,Z 371.568,A -85,B 0,C 180,E1 -20802.402,E2 -20802.402} C_VEL
LIN {X 0,Y 211.795,Z 375.483,A -85,B 0,C 180,E1 -20805.788,E2 -20805.788} C_VEL
LIN {X 0,Y 211.308,Z 378.167,A -85,B 0,C 180,E1 -20809.426,E2 -20809.426} C_VEL
LIN {X 0,Y 211.227,Z 378.983,A -85,B 0,C 180,E1 -20811.469,E2 -20811.469} C_VEL
LIN {X 0,Y 211.272,Z 379.365,A -85,B 0,C 180,E1 -20813.527,E2 -20813.527} C_VEL
LIN {X 0,Y 211.574,Z 379.161,A -85,B 0,C 180,E1 -20816.254,E2 -20816.254} C_VEL
LIN {X 0,Y 212.342,Z 377.709,A -85,B 0,C 180,E1 -20819.766,E2 -20819.766} C_VEL
LIN {X 0,Y 213.433,Z 375.219,A -85,B 0,C 180,E1 -20822.91,E2 -20822.91} C_VEL
LIN {X 0,Y 215.007,Z 371.511,A -85,B 0,C 180,E1 -20826.041,E2 -20826.041} C_VEL
LIN {X 0,Y 217.34,Z 365.73,A -85,B 0,C 180,E1 -20829.494,E2 -20829.494} C_VEL
LIN {X 0,Y 219.715,Z 359.743,A -85,B 0,C 180,E1 -20832.2,E2 -20832.2} C_VEL
LIN {X 0,Y 222.335,Z 352.775,A -85,B 0,C 180,E1 -20834.694,E2 -20834.694} C_VEL
LIN {X 0,Y 225.396,Z 343.951,A -85,B 0,C 180,E1 -20837.192,E2 -20837.192} C_VEL
LIN {X 0,Y 228.646,Z 333.542,A -85,B 0,C 180,E1 -20839.487,E2 -20839.487} C_VEL
LIN {X 0,Y 231.626,Z 322.553,A -85,B 0,C 180,E1 -20841.38,E2 -20841.38} C_VEL
LIN {X 0,Y 234.151,Z 311.594,A -85,B 0,C 180,E1 -20842.835,E2 -20842.835} C_VEL
LIN {X 0,Y 236.384,Z 299.105,A -85,B 0,C 180,E1 -20844.113,E2 -20844.113} C_VEL
LIN {X 0,Y 238.041,Z 286.279,A -85,B 0,C 180,E1 -20845.061,E2 -20845.061} C_VEL
LIN {X 0,Y 239.188,Z 273.649,A -85,B 0,C 180,E1 -20845.647,E2 -20845.647} C_VEL
LIN {X 0,Y 241.93,Z 220.633,A -85,B 0,C 180,E1 -20847.248,E2 -20847.248} C_VEL
LIN {X 0,Y 236.622,Z 208.594,A -85,B 0,C 180,E1 -20848.852,E2 -20848.852} C_VEL
LIN {X 0,Y 230.418,Z 196.797,A -85,B 0,C 180,E1 -20850.792,E2 -20850.792} C_VEL
LIN {X 0,Y 225.03,Z 188.527,A -85,B 0,C 180,E1 -20852.548,E2 -20852.548} C_VEL
LIN {X 0,Y 222.696,Z 185.218,A -85,B 0,C 180,E1 -20853.345,E2 -20853.345} C_VEL
LIN {X 0,Y 219.823,Z 181.081,A -85,B 0,C 180,E1 -20854.369,E2 -20854.369} C_VEL
LIN {X 0,Y 217.645,Z 177.996,A -85,B 0,C 180,E1 -20855.181,E2 -20855.181} C_VEL
LIN {X 0,Y 216.895,Z 176.857,A -85,B 0,C 180,E1 -20855.473,E2 -20855.473} C_VEL
LIN {X 0,Y 214.857,Z 174.738,A -85,B 0,C 180,E1 -20856.239,E2 -20856.239} C_VEL
LIN {X 0,Y 213.866,Z 172.152,A -85,B 0,C 180,E1 -20856.713,E2 -20856.713} C_VEL
LIN {X 0,Y 213.846,Z 171.848,A -85,B 0,C 180,E1 -20856.775,E2 -20856.775} C_VEL
LIN {X 0,Y 213.927,Z 171.829,A -85,B 0,C 180,E1 -20862.311,E2 -20862.311} C_VEL
LIN {X 0,Y 213.944,Z 171.824,A -85,B 0,C 180,E1 -20866.708,E2 -20866.708} C_VEL
LIN {X 0,Y 214.136,Z 171.798,A -85,B 0,C 180,E1 -20870.557,E2 -20870.557} C_VEL
LIN {X 0,Y 214.087,Z 171.809,A -85,B 0,C 180,E1 -20874.35,E2 -20874.35} C_VEL
LIN {X 0,Y 214.442,Z 171.769,A -85,B 0,C 180,E1 -20878.123,E2 -20878.123} C_VEL
LIN {X 0,Y 214.538,Z 171.743,A -85,B 0,C 180,E1 -20880.002,E2 -20880.002} C_VEL
LIN {X 0,Y 214.409,Z 171.761,A -85,B 0,C 180,E1 -20881.88,E2 -20881.88} C_VEL
LIN {X 0,Y 214.187,Z 171.795,A -85,B 0,C 180,E1 -20887.543,E2 -20887.543} C_VEL
LIN {X 0,Y 213.993,Z 171.809,A -85,B 0,C 180,E1 -20891.366,E2 -20891.366} C_VEL
LIN {X 0,Y 213.896,Z 171.829,A -85,B 0,C 180,E1 -20895.241,E2 -20895.241} C_VEL
LIN {X 0,Y 213.796,Z 171.855,A -85,B 0,C 180,E1 -20899.193,E2 -20899.193} C_VEL
LIN {X 0,Y 213.786,Z 171.852,A -85,B 0,C 180,E1 -20903.236,E2 -20903.236} C_VEL
LIN {X 0,Y 213.787,Z 171.847,A -85,B 0,C 180,E1 -20907.428,E2 -20907.428} C_VEL
LIN {X 0,Y 213.761,Z 171.851,A -85,B 0,C 180,E1 -20911.74,E2 -20911.74} C_VEL
LIN {X 0,Y 213.743,Z 171.862,A -85,B 0,C 180,E1 -20916.29,E2 -20916.29} C_VEL
LIN {X 0,Y 213.714,Z 171.857,A -85,B 0,C 180,E1 -20917.912,E2 -20917.912} C_VEL
LIN {X 0,Y 213.116,Z 172.326,A -85,B 0,C 180,E1 -20918.957,E2 -20918.957} C_VEL
LIN {X 0,Y 210.804,Z 174.473,A -85,B 0,C 180,E1 -20920.565,E2 -20920.565} C_VEL
LIN {X 0,Y 208.745,Z 177.366,A -85,B 0,C 180,E1 -20922.163,E2 -20922.163} C_VEL
LIN {X 0,Y 208.595,Z 179.001,A -85,B 0,C 180,E1 -20923.179,E2 -20923.179} C_VEL
LIN {X 0,Y 208.909,Z 179.78,A -85,B 0,C 180,E1 -20923.521,E2 -20923.521} C_VEL
LIN {X 0,Y 211.948,Z 184.513,A -85,B 0,C 180,E1 -20924.857,E2 -20924.857} C_VEL
LIN {X 0,Y 213.682,Z 187.298,A -85,B 0,C 180,E1 -20925.59,E2 -20925.59} C_VEL
LIN {X 0,Y 216.653,Z 192.039,A -85,B 0,C 180,E1 -20926.772,E2 -20926.772} C_VEL
LIN {X 0,Y 222.056,Z 201.13,A -85,B 0,C 180,E1 -20928.778,E2 -20928.778} C_VEL
LIN {X 0,Y 227.966,Z 212.835,A -85,B 0,C 180,E1 -20930.857,E2 -20930.857} C_VEL
LIN {X 0,Y 233.853,Z 226.714,A -85,B 0,C 180,E1 -20932.829,E2 -20932.829} C_VEL
LIN {X 0,Y 235.607,Z 241.593,A -85,B 0,C 180,E1 -20933.83,E2 -20933.83} C_VEL
LIN {X 0,Y 232.907,Z 290.147,A -85,B 0,C 180,E1 -20935.347,E2 -20935.347} C_VEL
LIN {X 0,Y 231.331,Z 303.627,A -85,B 0,C 180,E1 -20936.066,E2 -20936.066} C_VEL
LIN {X 0,Y 229.151,Z 315.937,A -85,B 0,C 180,E1 -20937.017,E2 -20937.017} C_VEL
LIN {X 0,Y 226.601,Z 327.011,A -85,B 0,C 180,E1 -20938.18,E2 -20938.18} C_VEL
LIN {X 0,Y 223.638,Z 338.532,A -85,B 0,C 180,E1 -20939.814,E2 -20939.814} C_VEL
LIN {X 0,Y 220.476,Z 348.961,A -85,B 0,C 180,E1 -20941.695,E2 -20941.695} C_VEL
LIN {X 0,Y 217.519,Z 357.528,A -85,B 0,C 180,E1 -20943.624,E2 -20943.624} C_VEL
LIN {X 0,Y 214.682,Z 365.449,A -85,B 0,C 180,E1 -20945.845,E2 -20945.845} C_VEL
LIN {X 0,Y 211.906,Z 373.229,A -85,B 0,C 180,E1 -20948.604,E2 -20948.604} C_VEL
LIN {X 0,Y 209.408,Z 379.495,A -85,B 0,C 180,E1 -20951.408,E2 -20951.408} C_VEL
LIN {X 0,Y 207.312,Z 384.504,A -85,B 0,C 180,E1 -20954.264,E2 -20954.264} C_VEL
LIN {X 0,Y 205.891,Z 388.402,A -85,B 0,C 180,E1 -20957.181,E2 -20957.181} C_VEL
LIN {X 0,Y 204.967,Z 391.292,A -85,B 0,C 180,E1 -20960.129,E2 -20960.129} C_VEL
LIN {X 0,Y 204.395,Z 393.671,A -85,B 0,C 180,E1 -20964.08,E2 -20964.08} C_VEL
LIN {X 0,Y 204.34,Z 394.28,A -85,B 0,C 180,E1 -20966.056,E2 -20966.056} C_VEL
LIN {X 0,Y 204.411,Z 394.462,A -85,B 0,C 180,E1 -20968.03,E2 -20968.03} C_VEL
LIN {X 0,Y 204.555,Z 394.236,A -85,B 0,C 180,E1 -20970,E2 -20970} C_VEL
LIN {X 0,Y 204.447,Z 393.606,A -85,B 0,C 180,E1 -20971.97,E2 -20971.97} C_VEL
LIN {X 0,Y 204.357,Z 392.434,A -85,B 0,C 180,E1 -20974.166,E2 -20974.166} C_VEL
LIN {X 0,Y 204.627,Z 389.166,A -85,B 0,C 180,E1 -20977.897,E2 -20977.897} C_VEL
LIN {X 0,Y 205.163,Z 385.411,A -85,B 0,C 180,E1 -20980.86,E2 -20980.86} C_VEL
LIN {X 0,Y 206.101,Z 380.51,A -85,B 0,C 180,E1 -20983.81,E2 -20983.81} C_VEL
LIN {X 0,Y 207.715,Z 374.333,A -85,B 0,C 180,E1 -20986.715,E2 -20986.715} C_VEL
LIN {X 0,Y 209.69,Z 366.623,A -85,B 0,C 180,E1 -20989.583,E2 -20989.583} C_VEL
LIN {X 0,Y 211.55,Z 358.695,A -85,B 0,C 180,E1 -20991.947,E2 -20991.947} C_VEL
LIN {X 0,Y 213.889,Z 349.023,A -85,B 0,C 180,E1 -20994.251,E2 -20994.251} C_VEL
LIN {X 0,Y 216.367,Z 338.304,A -85,B 0,C 180,E1 -20996.268,E2 -20996.268} C_VEL
LIN {X 0,Y 218.493,Z 327.948,A -85,B 0,C 180,E1 -20997.802,E2 -20997.802} C_VEL
LIN {X 0,Y 220.624,Z 315.582,A -85,B 0,C 180,E1 -20999.195,E2 -20999.195} C_VEL
LIN {X 0,Y 222.35,Z 302.62,A -85,B 0,C 180,E1 -21000.249,E2 -21000.249} C_VEL
LIN {X 0,Y 223.486,Z 290.181,A -85,B 0,C 180,E1 -21000.925,E2 -21000.925} C_VEL
LIN {X 0,Y 225.625,Z 237.656,A -85,B 0,C 180,E1 -21002.628,E2 -21002.628} C_VEL
LIN {X 0,Y 222.446,Z 214.011,A -85,B 0,C 180,E1 -21003.966,E2 -21003.966} C_VEL
LIN {X 0,Y 215.28,Z 195.891,A -85,B 0,C 180,E1 -21005.768,E2 -21005.768} C_VEL
LIN {X 0,Y 208.877,Z 181.539,A -85,B 0,C 180,E1 -21007.486,E2 -21007.486} C_VEL
LIN {X 0,Y 206.619,Z 172.737,A -85,B 0,C 180,E1 -21011.925,E2 -21011.925} C_VEL
LIN {X 0,Y 206.634,Z 172.747,A -85,B 0,C 180,E1 -21015.583,E2 -21015.583} C_VEL
LIN {X 0,Y 206.652,Z 172.747,A -85,B 0,C 180,E1 -21019.745,E2 -21019.745} C_VEL
LIN {X 0,Y 206.705,Z 172.74,A -85,B 0,C 180,E1 -21024.688,E2 -21024.688} C_VEL
LIN {X 0,Y 206.701,Z 172.739,A -85,B 0,C 180,E1 -21029.334,E2 -21029.334} C_VEL
LIN {X 0,Y 206.709,Z 172.736,A -85,B 0,C 180,E1 -21033.767,E2 -21033.767} C_VEL
LIN {X 0,Y 206.721,Z 172.734,A -85,B 0,C 180,E1 -21038.038,E2 -21038.038} C_VEL
LIN {X 0,Y 206.807,Z 172.724,A -85,B 0,C 180,E1 -21042.189,E2 -21042.189} C_VEL
LIN {X 0,Y 206.862,Z 172.717,A -85,B 0,C 180,E1 -21046.24,E2 -21046.24} C_VEL
LIN {X 0,Y 207.082,Z 172.674,A -85,B 0,C 180,E1 -21050.229,E2 -21050.229} C_VEL
LIN {X 0,Y 207.042,Z 172.681,A -85,B 0,C 180,E1 -21054.154,E2 -21054.154} C_VEL
LIN {X 0,Y 207.348,Z 172.658,A -85,B 0,C 180,E1 -21058.056,E2 -21058.056} C_VEL
LIN {X 0,Y 207.484,Z 172.633,A -85,B 0,C 180,E1 -21059.998,E2 -21059.998} C_VEL
LIN {X 0,Y 207.346,Z 172.635,A -85,B 0,C 180,E1 -21061.941,E2 -21061.941} C_VEL
LIN {X 0,Y 207.13,Z 172.68,A -85,B 0,C 180,E1 -21067.799,E2 -21067.799} C_VEL
LIN {X 0,Y 206.904,Z 172.707,A -85,B 0,C 180,E1 -21071.758,E2 -21071.758} C_VEL
LIN {X 0,Y 206.8,Z 172.697,A -85,B 0,C 180,E1 -21075.774,E2 -21075.774} C_VEL
LIN {X 0,Y 206.712,Z 172.732,A -85,B 0,C 180,E1 -21079.874,E2 -21079.874} C_VEL
LIN {X 0,Y 206.699,Z 172.73,A -85,B 0,C 180,E1 -21084.078,E2 -21084.078} C_VEL
LIN {X 0,Y 206.685,Z 172.718,A -85,B 0,C 180,E1 -21088.426,E2 -21088.426} C_VEL
LIN {X 0,Y 206.692,Z 172.738,A -85,B 0,C 180,E1 -21092.957,E2 -21092.957} C_VEL
LIN {X 0,Y 206.698,Z 172.731,A -85,B 0,C 180,E1 -21095.309,E2 -21095.309} C_VEL
LIN {X 0,Y 206.644,Z 172.738,A -85,B 0,C 180,E1 -21100.253,E2 -21100.253} C_VEL
LIN {X 0,Y 206.626,Z 172.746,A -85,B 0,C 180,E1 -21104.415,E2 -21104.415} C_VEL
LIN {X 0,Y 206.627,Z 172.737,A -85,B 0,C 180,E1 -21108.439,E2 -21108.439} C_VEL
LIN {X 0,Y 206.664,Z 172.744,A -85,B 0,C 180,E1 -21112.256,E2 -21112.256} C_VEL
LIN {X 0,Y 206.69,Z 172.738,A -85,B 0,C 180,E1 -21117.04,E2 -21117.04} C_VEL
LIN {X 0,Y 206.703,Z 172.731,A -85,B 0,C 180,E1 -21122.126,E2 -21122.126} C_VEL
LIN {X 0,Y 206.721,Z 172.722,A -85,B 0,C 180,E1 -21126.621,E2 -21126.621} C_VEL
LIN {X 0,Y 206.797,Z 172.728,A -85,B 0,C 180,E1 -21132.189,E2 -21132.189} C_VEL
LIN {X 0,Y 206.819,Z 172.772,A -85,B 0,C 180,E1 -21134.442,E2 -21134.442} C_VEL
LIN {X 0,Y 207.797,Z 175.504,A -85,B 0,C 180,E1 -21134.732,E2 -21134.732} C_VEL
LIN {X 0,Y 211.338,Z 181.538,A -85,B 0,C 180,E1 -21135.596,E2 -21135.596} C_VEL
LIN {X 0,Y 219.336,Z 196.298,A -85,B 0,C 180,E1 -21137.49,E2 -21137.49} C_VEL
LIN {X 0,Y 226.673,Z 215.161,A -85,B 0,C 180,E1 -21139.278,E2 -21139.278} C_VEL
LIN {X 0,Y 223.793,Z 275.899,A -85,B 0,C 180,E1 -21141.193,E2 -21141.193} C_VEL
LIN {X 0,Y 222.563,Z 289.876,A -85,B 0,C 180,E1 -21142.002,E2 -21142.002} C_VEL
LIN {X 0,Y 221.185,Z 301.815,A -85,B 0,C 180,E1 -21143.042,E2 -21143.042} C_VEL
LIN {X 0,Y 219.342,Z 313.964,A -85,B 0,C 180,E1 -21144.484,E2 -21144.484} C_VEL
LIN {X 0,Y 217.068,Z 325.654,A -85,B 0,C 180,E1 -21146.287,E2 -21146.287} C_VEL
LIN {X 0,Y 214.761,Z 336.151,A -85,B 0,C 180,E1 -21148.359,E2 -21148.359} C_VEL
LIN {X 0,Y 212.26,Z 346.391,A -85,B 0,C 180,E1 -21150.948,E2 -21150.948} C_VEL
LIN {X 0,Y 210.233,Z 354.172,A -85,B 0,C 180,E1 -21153.412,E2 -21153.412} C_VEL
LIN {X 0,Y 208.305,Z 361.461,A -85,B 0,C 180,E1 -21156.295,E2 -21156.295} C_VEL
LIN {X 0,Y 206.656,Z 367.763,A -85,B 0,C 180,E1 -21159.528,E2 -21159.528} C_VEL
LIN {X 0,Y 205.452,Z 372.653,A -85,B 0,C 180,E1 -21162.847,E2 -21162.847} C_VEL
LIN {X 0,Y 204.651,Z 375.965,A -85,B 0,C 180,E1 -21165.946,E2 -21165.946} C_VEL
LIN {X 0,Y 204.333,Z 377.592,A -85,B 0,C 180,E1 -21168.032,E2 -21168.032} C_VEL
LIN {X 0,Y 204.125,Z 379.257,A -85,B 0,C 180,E1 -21171.632,E2 -21171.632} C_VEL
LIN {X 0,Y 204.231,Z 379.674,A -85,B 0,C 180,E1 -21174.39,E2 -21174.39} C_VEL
LIN {X 0,Y 204.564,Z 379.384,A -85,B 0,C 180,E1 -21176.719,E2 -21176.719} C_VEL
LIN {X 0,Y 204.924,Z 378.739,A -85,B 0,C 180,E1 -21178.694,E2 -21178.694} C_VEL
LIN {X 0,Y 205.739,Z 377.196,A -85,B 0,C 180,E1 -21181.355,E2 -21181.355} C_VEL
LIN {X 0,Y 207.384,Z 373.647,A -85,B 0,C 180,E1 -21185.177,E2 -21185.177} C_VEL
LIN {X 0,Y 209.38,Z 369.196,A -85,B 0,C 180,E1 -21188.387,E2 -21188.387} C_VEL
LIN {X 0,Y 211.863,Z 363.275,A -85,B 0,C 180,E1 -21191.563,E2 -21191.563} C_VEL
LIN {X 0,Y 214.87,Z 355.965,A -85,B 0,C 180,E1 -21194.555,E2 -21194.555} C_VEL
LIN {X 0,Y 217.861,Z 348.018,A -85,B 0,C 180,E1 -21197.081,E2 -21197.081} C_VEL
LIN {X 0,Y 221.05,Z 338.849,A -85,B 0,C 180,E1 -21199.382,E2 -21199.382} C_VEL
LIN {X 0,Y 224.354,Z 327.945,A -85,B 0,C 180,E1 -21201.548,E2 -21201.548} C_VEL
LIN {X 0,Y 227.156,Z 317.255,A -85,B 0,C 180,E1 -21203.182,E2 -21203.182} C_VEL
LIN {X 0,Y 229.607,Z 305.705,A -85,B 0,C 180,E1 -21204.56,E2 -21204.56} C_VEL
LIN {X 0,Y 231.556,Z 294.042,A -85,B 0,C 180,E1 -21205.606,E2 -21205.606} C_VEL
LIN {X 0,Y 233.034,Z 281.292,A -85,B 0,C 180,E1 -21206.422,E2 -21206.422} C_VEL
LIN {X 0,Y 234.186,Z 265.862,A -85,B 0,C 180,E1 -21206.975,E2 -21206.975} C_VEL
LIN {X 0,Y 236.444,Z 222.877,A -85,B 0,C 180,E1 -21208.291,E2 -21208.291} C_VEL
LIN {X 0,Y 230.738,Z 210.072,A -85,B 0,C 180,E1 -21210.119,E2 -21210.119} C_VEL
LIN {X 0,Y 225.461,Z 200.328,A -85,B 0,C 180,E1 -21211.872,E2 -21211.872} C_VEL
LIN {X 0,Y 219.664,Z 191.288,A -85,B 0,C 180,E1 -21213.895,E2 -21213.895} C_VEL
LIN {X 0,Y 215.655,Z 185.757,A -85,B 0,C 180,E1 -21215.387,E2 -21215.387} C_VEL
LIN {X 0,Y 213.507,Z 182.586,A -85,B 0,C 180,E1 -21216.247,E2 -21216.247} C_VEL
LIN {X 0,Y 211.098,Z 179.549,A -85,B 0,C 180,E1 -21217.235,E2 -21217.235} C_VEL
LIN {X 0,Y 210.183,Z 177.949,A -85,B 0,C 180,E1 -21217.648,E2 -21217.648} C_VEL
LIN {X 0,Y 207.968,Z 175.884,A -85,B 0,C 180,E1 -21218.57,E2 -21218.57} C_VEL
LIN {X 0,Y 206.915,Z 173.518,A -85,B 0,C 180,E1 -21219.108,E2 -21219.108} C_VEL
LIN {X 0,Y 206.755,Z 172.725,A -85,B 0,C 180,E1 -21219.221,E2 -21219.221} C_VEL
LIN {X 0,Y 206.867,Z 172.709,A -85,B 0,C 180,E1 -21222.198,E2 -21222.198} C_VEL
LIN {X 0,Y 206.886,Z 172.703,A -85,B 0,C 180,E1 -21226.245,E2 -21226.245} C_VEL
LIN {X 0,Y 207.079,Z 172.679,A -85,B 0,C 180,E1 -21230.232,E2 -21230.232} C_VEL
LIN {X 0,Y 207.049,Z 172.687,A -85,B 0,C 180,E1 -21234.157,E2 -21234.157} C_VEL
LIN {X 0,Y 207.378,Z 172.648,A -85,B 0,C 180,E1 -21238.059,E2 -21238.059} C_VEL
LIN {X 0,Y 207.503,Z 172.618,A -85,B 0,C 180,E1 -21240.002,E2 -21240.002} C_VEL
LIN {X 0,Y 207.049,Z 172.686,A -85,B 0,C 180,E1 -21243.894,E2 -21243.894} C_VEL
LIN {X 0,Y 207.131,Z 172.677,A -85,B 0,C 180,E1 -21247.802,E2 -21247.802} C_VEL
LIN {X 0,Y 206.915,Z 172.692,A -85,B 0,C 180,E1 -21251.76,E2 -21251.76} C_VEL
LIN {X 0,Y 206.824,Z 172.706,A -85,B 0,C 180,E1 -21255.776,E2 -21255.776} C_VEL
LIN {X 0,Y 206.716,Z 172.73,A -85,B 0,C 180,E1 -21259.877,E2 -21259.877} C_VEL
LIN {X 0,Y 206.723,Z 172.735,A -85,B 0,C 180,E1 -21264.079,E2 -21264.079} C_VEL
LIN {X 0,Y 206.689,Z 172.74,A -85,B 0,C 180,E1 -21268.429,E2 -21268.429} C_VEL
LIN {X 0,Y 206.696,Z 172.737,A -85,B 0,C 180,E1 -21272.96,E2 -21272.96} C_VEL
LIN {X 0,Y 206.702,Z 172.73,A -85,B 0,C 180,E1 -21275.312,E2 -21275.312} C_VEL
LIN {X 0,Y 206.695,Z 172.885,A -85,B 0,C 180,E1 -21278.66,E2 -21278.66} C_VEL
LIN {X 0,Y 208.595,Z 179.001,A -85,B 0,C 180,E1 -21283.179,E2 -21283.179} C_VEL
LIN {X 0,Y 209.548,Z 180.395,A -85,B 0,C 180,E1 -21283.786,E2 -21283.786} C_VEL
LIN {X 0,Y 211.266,Z 183.765,A -85,B 0,C 180,E1 -21284.582,E2 -21284.582} C_VEL
LIN {X 0,Y 213.094,Z 190.559,A -85,B 0,C 180,E1 -21285.578,E2 -21285.578} C_VEL
LIN {X 0,Y 215.292,Z 199.806,A -85,B 0,C 180,E1 -21286.724,E2 -21286.724} C_VEL
LIN {X 0,Y 217.288,Z 204.59,A -85,B 0,C 180,E1 -21287.611,E2 -21287.611} C_VEL
LIN {X 0,Y 222.753,Z 215.419,A -85,B 0,C 180,E1 -21289.656,E2 -21289.656} C_VEL
LIN {X 0,Y 227.678,Z 226.889,A -85,B 0,C 180,E1 -21291.424,E2 -21291.424} C_VEL
LIN {X 0,Y 228.891,Z 230.088,A -85,B 0,C 180,E1 -21291.857,E2 -21291.857} C_VEL
LIN {X 0,Y 230.221,Z 242.599,A -85,B 0,C 180,E1 -21292.708,E2 -21292.708} C_VEL
LIN {X 0,Y 227.498,Z 289.574,A -85,B 0,C 180,E1 -21294.195,E2 -21294.195} C_VEL
LIN {X 0,Y 225.864,Z 303.147,A -85,B 0,C 180,E1 -21294.923,E2 -21294.923} C_VEL
LIN {X 0,Y 223.489,Z 316.047,A -85,B 0,C 180,E1 -21295.934,E2 -21295.934} C_VEL
LIN {X 0,Y 220.638,Z 327.807,A -85,B 0,C 180,E1 -21297.214,E2 -21297.214} C_VEL
LIN {X 0,Y 217.571,Z 339.135,A -85,B 0,C 180,E1 -21298.88,E2 -21298.88} C_VEL
LIN {X 0,Y 214.277,Z 349.407,A -85,B 0,C 180,E1 -21300.799,E2 -21300.799} C_VEL
LIN {X 0,Y 211.197,Z 357.841,A -85,B 0,C 180,E1 -21302.771,E2 -21302.771} C_VEL
LIN {X 0,Y 207.666,Z 367.013,A -85,B 0,C 180,E1 -21305.508,E2 -21305.508} C_VEL
LIN {X 0,Y 204.811,Z 374.428,A -85,B 0,C 180,E1 -21308.354,E2 -21308.354} C_VEL
LIN {X 0,Y 202.655,Z 379.507,A -85,B 0,C 180,E1 -21310.764,E2 -21310.764} C_VEL
LIN {X 0,Y 200.48,Z 384.458,A -85,B 0,C 180,E1 -21313.713,E2 -21313.713} C_VEL
LIN {X 0,Y 198.923,Z 388.301,A -85,B 0,C 180,E1 -21316.724,E2 -21316.724} C_VEL
LIN {X 0,Y 197.95,Z 391.14,A -85,B 0,C 180,E1 -21319.775,E2 -21319.775} C_VEL
LIN {X 0,Y 197.31,Z 393.47,A -85,B 0,C 180,E1 -21323.866,E2 -21323.866} C_VEL
LIN {X 0,Y 197.255,Z 394.064,A -85,B 0,C 180,E1 -21326.058,E2 -21326.058} C_VEL
LIN {X 0,Y 197.47,Z 393.942,A -85,B 0,C 180,E1 -21330,E2 -21330} C_VEL
LIN {X 0,Y 197.345,Z 393.288,A -85,B 0,C 180,E1 -21332.041,E2 -21332.041} C_VEL
LIN {X 0,Y 197.255,Z 392.227,A -85,B 0,C 180,E1 -21334.087,E2 -21334.087} C_VEL
LIN {X 0,Y 197.344,Z 390.705,A -85,B 0,C 180,E1 -21336.134,E2 -21336.134} C_VEL
LIN {X 0,Y 197.72,Z 387.613,A -85,B 0,C 180,E1 -21339.205,E2 -21339.205} C_VEL
LIN {X 0,Y 198.467,Z 383.435,A -85,B 0,C 180,E1 -21342.268,E2 -21342.268} C_VEL
LIN {X 0,Y 199.7,Z 378.058,A -85,B 0,C 180,E1 -21345.305,E2 -21345.305} C_VEL
LIN {X 0,Y 201.45,Z 371.305,A -85,B 0,C 180,E1 -21348.3,E2 -21348.3} C_VEL
LIN {X 0,Y 202.934,Z 365.925,A -85,B 0,C 180,E1 -21350.263,E2 -21350.263} C_VEL
LIN {X 0,Y 204.905,Z 357.898,A -85,B 0,C 180,E1 -21352.698,E2 -21352.698} C_VEL
LIN {X 0,Y 207.37,Z 348.116,A -85,B 0,C 180,E1 -21355.065,E2 -21355.065} C_VEL
LIN {X 0,Y 209.959,Z 337.258,A -85,B 0,C 180,E1 -21357.135,E2 -21357.135} C_VEL
LIN {X 0,Y 212.206,Z 326.678,A -85,B 0,C 180,E1 -21358.701,E2 -21358.701} C_VEL
LIN {X 0,Y 214.449,Z 313.967,A -85,B 0,C 180,E1 -21360.122,E2 -21360.122} C_VEL
LIN {X 0,Y 216.136,Z 301.293,A -85,B 0,C 180,E1 -21361.146,E2 -21361.146} C_VEL
LIN {X 0,Y 217.275,Z 288.15,A -85,B 0,C 180,E1 -21361.832,E2 -21361.832} C_VEL
LIN {X 0,Y 219.402,Z 238.88,A -85,B 0,C 180,E1 -21363.45,E2 -21363.45} C_VEL
LIN {X 0,Y 216.446,Z 216.378,A -85,B 0,C 180,E1 -21364.767,E2 -21364.767} C_VEL
LIN {X 0,Y 209.485,Z 198.672,A -85,B 0,C 180,E1 -21366.611,E2 -21366.611} C_VEL
LIN {X 0,Y 203.034,Z 184.673,A -85,B 0,C 180,E1 -21368.338,E2 -21368.338} C_VEL
LIN {X 0,Y 201.545,Z 181.283,A -85,B 0,C 180,E1 -21368.813,E2 -21368.813} C_VEL
LIN {X 0,Y 199.572,Z 173.615,A -85,B 0,C 180,E1 -21372.962,E2 -21372.962} C_VEL
LIN {X 0,Y 199.575,Z 173.627,A -85,B 0,C 180,E1 -21378.002,E2 -21378.002} C_VEL
LIN {X 0,Y 199.602,Z 173.625,A -85,B 0,C 180,E1 -21380.772,E2 -21380.772} C_VEL
LIN {X 0,Y 199.615,Z 173.622,A -85,B 0,C 180,E1 -21385.712,E2 -21385.712} C_VEL
LIN {X 0,Y 199.691,Z 173.612,A -85,B 0,C 180,E1 -21388.133,E2 -21388.133} C_VEL
LIN {X 0,Y 199.648,Z 173.617,A -85,B 0,C 180,E1 -21392.764,E2 -21392.764} C_VEL
LIN {X 0,Y 199.683,Z 173.611,A -85,B 0,C 180,E1 -21397.221,E2 -21397.221} C_VEL
LIN {X 0,Y 199.75,Z 173.602,A -85,B 0,C 180,E1 -21401.802,E2 -21401.802} C_VEL
LIN {X 0,Y 199.8,Z 173.595,A -85,B 0,C 180,E1 -21405.744,E2 -21405.744} C_VEL
LIN {X 0,Y 200.027,Z 173.555,A -85,B 0,C 180,E1 -21409.88,E2 -21409.88} C_VEL
LIN {X 0,Y 200.005,Z 173.556,A -85,B 0,C 180,E1 -21413.947,E2 -21413.947} C_VEL
LIN {X 0,Y 200.29,Z 173.537,A -85,B 0,C 180,E1 -21417.987,E2 -21417.987} C_VEL
LIN {X 0,Y 200.451,Z 173.509,A -85,B 0,C 180,E1 -21419.998,E2 -21419.998} C_VEL
LIN {X 0,Y 199.99,Z 173.544,A -85,B 0,C 180,E1 -21424.029,E2 -21424.029} C_VEL
LIN {X 0,Y 200.077,Z 173.56,A -85,B 0,C 180,E1 -21428.075,E2 -21428.075} C_VEL
LIN {X 0,Y 199.854,Z 173.582,A -85,B 0,C 180,E1 -21432.179,E2 -21432.179} C_VEL
LIN {X 0,Y 199.741,Z 173.576,A -85,B 0,C 180,E1 -21436.347,E2 -21436.347} C_VEL
LIN {X 0,Y 199.642,Z 173.615,A -85,B 0,C 180,E1 -21440.61,E2 -21440.61} C_VEL
LIN {X 0,Y 199.624,Z 173.607,A -85,B 0,C 180,E1 -21444.989,E2 -21444.989} C_VEL
LIN {X 0,Y 199.606,Z 173.606,A -85,B 0,C 180,E1 -21449.531,E2 -21449.531} C_VEL
LIN {X 0,Y 199.664,Z 173.613,A -85,B 0,C 180,E1 -21452.35,E2 -21452.35} C_VEL
LIN {X 0,Y 199.613,Z 173.603,A -85,B 0,C 180,E1 -21456.763,E2 -21456.763} C_VEL
LIN {X 0,Y 199.591,Z 173.605,A -85,B 0,C 180,E1 -21459.33,E2 -21459.33} C_VEL
LIN {X 0,Y 199.563,Z 173.627,A -85,B 0,C 180,E1 -21462.305,E2 -21462.305} C_VEL
LIN {X 0,Y 199.572,Z 173.619,A -85,B 0,C 180,E1 -21465.226,E2 -21465.226} C_VEL
LIN {X 0,Y 199.566,Z 173.613,A -85,B 0,C 180,E1 -21468.001,E2 -21468.001} C_VEL
LIN {X 0,Y 199.593,Z 173.626,A -85,B 0,C 180,E1 -21470.771,E2 -21470.771} C_VEL
LIN {X 0,Y 199.606,Z 173.613,A -85,B 0,C 180,E1 -21475.711,E2 -21475.711} C_VEL
LIN {X 0,Y 199.681,Z 173.614,A -85,B 0,C 180,E1 -21478.133,E2 -21478.133} C_VEL
LIN {X 0,Y 199.63,Z 173.615,A -85,B 0,C 180,E1 -21482.763,E2 -21482.763} C_VEL
LIN {X 0,Y 199.665,Z 173.601,A -85,B 0,C 180,E1 -21487.22,E2 -21487.22} C_VEL
LIN {X 0,Y 199.743,Z 173.603,A -85,B 0,C 180,E1 -21492.959,E2 -21492.959} C_VEL
LIN {X 0,Y 199.755,Z 173.834,A -85,B 0,C 180,E1 -21493.162,E2 -21493.162} C_VEL
LIN {X 0,Y 200.868,Z 176.634,A -85,B 0,C 180,E1 -21493.503,E2 -21493.503} C_VEL
LIN {X 0,Y 202.327,Z 178.943,A -85,B 0,C 180,E1 -21493.882,E2 -21493.882} C_VEL
LIN {X 0,Y 211.291,Z 194.925,A -85,B 0,C 180,E1 -21496.141,E2 -21496.141} C_VEL
LIN {X 0,Y 215.035,Z 202.655,A -85,B 0,C 180,E1 -21497.068,E2 -21497.068} C_VEL
LIN {X 0,Y 220.379,Z 216.675,A -85,B 0,C 180,E1 -21498.438,E2 -21498.438} C_VEL
LIN {X 0,Y 217.457,Z 276.645,A -85,B 0,C 180,E1 -21500.389,E2 -21500.389} C_VEL
LIN {X 0,Y 216.231,Z 289.934,A -85,B 0,C 180,E1 -21501.177,E2 -21501.177} C_VEL
LIN {X 0,Y 214.786,Z 301.93,A -85,B 0,C 180,E1 -21502.242,E2 -21502.242} C_VEL
LIN {X 0,Y 213.013,Z 313.318,A -85,B 0,C 180,E1 -21503.606,E2 -21503.606} C_VEL
LIN {X 0,Y 210.663,Z 325.159,A -85,B 0,C 180,E1 -21505.454,E2 -21505.454} C_VEL
LIN {X 0,Y 208.23,Z 335.82,A -85,B 0,C 180,E1 -21507.582,E2 -21507.582} C_VEL
LIN {X 0,Y 205.861,Z 345.335,A -85,B 0,C 180,E1 -21510,E2 -21510} C_VEL
LIN {X 0,Y 203.328,Z 354.575,A -85,B 0,C 180,E1 -21512.971,E2 -21512.971} C_VEL
LIN {X 0,Y 201.284,Z 361.967,A -85,B 0,C 180,E1 -21516.012,E2 -21516.012} C_VEL
LIN {X 0,Y 199.532,Z 368.497,A -85,B 0,C 180,E1 -21519.532,E2 -21519.532} C_VEL
LIN {X 0,Y 198.205,Z 373.699,A -85,B 0,C 180,E1 -21523.325,E2 -21523.325} C_VEL
LIN {X 0,Y 197.44,Z 376.782,A -85,B 0,C 180,E1 -21526.544,E2 -21526.544} C_VEL
LIN {X 0,Y 197.172,Z 378.229,A -85,B 0,C 180,E1 -21528.711,E2 -21528.711} C_VEL
LIN {X 0,Y 197.057,Z 379.573,A -85,B 0,C 180,E1 -21531.99,E2 -21531.99} C_VEL
LIN {X 0,Y 197.233,Z 379.895,A -85,B 0,C 180,E1 -21535.315,E2 -21535.315} C_VEL
LIN {X 0,Y 197.6,Z 379.541,A -85,B 0,C 180,E1 -21537.54,E2 -21537.54} C_VEL
LIN {X 0,Y 198.096,Z 378.689,A -85,B 0,C 180,E1 -21539.781,E2 -21539.781} C_VEL
LIN {X 0,Y 198.861,Z 377.341,A -85,B 0,C 180,E1 -21542.013,E2 -21542.013} C_VEL
LIN {X 0,Y 200.345,Z 374.372,A -85,B 0,C 180,E1 -21545.353,E2 -21545.353} C_VEL
LIN {X 0,Y 202.411,Z 370.115,A -85,B 0,C 180,E1 -21548.681,E2 -21548.681} C_VEL
LIN {X 0,Y 204.962,Z 364.387,A -85,B 0,C 180,E1 -21551.962,E2 -21551.962} C_VEL
LIN {X 0,Y 208.185,Z 357.016,A -85,B 0,C 180,E1 -21555.148,E2 -21555.148} C_VEL
LIN {X 0,Y 211.185,Z 349.649,A -85,B 0,C 180,E1 -21557.632,E2 -21557.632} C_VEL
LIN {X 0,Y 214.428,Z 340.824,A -85,B 0,C 180,E1 -21560.007,E2 -21560.007} C_VEL
LIN {X 0,Y 217.821,Z 330.426,A -85,B 0,C 180,E1 -21562.193,E2 -21562.193} C_VEL
LIN {X 0,Y 220.761,Z 320.166,A -85,B 0,C 180,E1 -21563.883,E2 -21563.883} C_VEL
LIN {X 0,Y 223.499,Z 308.577,A -85,B 0,C 180,E1 -21565.379,E2 -21565.379} C_VEL
LIN {X 0,Y 225.645,Z 297.027,A -85,B 0,C 180,E1 -21566.495,E2 -21566.495} C_VEL
LIN {X 0,Y 227.357,Z 283.756,A -85,B 0,C 180,E1 -21567.424,E2 -21567.424} C_VEL
LIN {X 0,Y 228.437,Z 271.615,A -85,B 0,C 180,E1 -21567.943,E2 -21567.943} C_VEL
LIN {X 0,Y 231.136,Z 225.517,A -85,B 0,C 180,E1 -21569.344,E2 -21569.344} C_VEL
LIN {X 0,Y 226.105,Z 213.956,A -85,B 0,C 180,E1 -21571.073,E2 -21571.073} C_VEL
LIN {X 0,Y 220.758,Z 203.976,A -85,B 0,C 180,E1 -21572.952,E2 -21572.952} C_VEL
LIN {X 0,Y 215.458,Z 195.884,A -85,B 0,C 180,E1 -21574.912,E2 -21574.912} C_VEL
LIN {X 0,Y 210.083,Z 188.099,A -85,B 0,C 180,E1 -21577.093,E2 -21577.093} C_VEL
LIN {X 0,Y 207.551,Z 184.595,A -85,B 0,C 180,E1 -21578.199,E2 -21578.199} C_VEL
LIN {X 0,Y 204.391,Z 180.762,A -85,B 0,C 180,E1 -21579.628,E2 -21579.628} C_VEL
LIN {X 0,Y 203.31,Z 178.918,A -85,B 0,C 180,E1 -21580.174,E2 -21580.174} C_VEL
LIN {X 0,Y 201.002,Z 176.817,A -85,B 0,C 180,E1 -21581.272,E2 -21581.272} C_VEL
LIN {X 0,Y 199.93,Z 174.309,A -85,B 0,C 180,E1 -21581.917,E2 -21581.917} C_VEL
LIN {X 0,Y 199.825,Z 173.587,A -85,B 0,C 180,E1 -21582.026,E2 -21582.026} C_VEL
LIN {X 0,Y 199.827,Z 173.585,A -85,B 0,C 180,E1 -21585.749,E2 -21585.749} C_VEL
LIN {X 0,Y 200.022,Z 173.561,A -85,B 0,C 180,E1 -21589.883,E2 -21589.883} C_VEL
LIN {X 0,Y 200.011,Z 173.565,A -85,B 0,C 180,E1 -21593.951,E2 -21593.951} C_VEL
LIN {X 0,Y 200.317,Z 173.527,A -85,B 0,C 180,E1 -21597.991,E2 -21597.991} C_VEL
LIN {X 0,Y 200.467,Z 173.494,A -85,B 0,C 180,E1 -21600.002,E2 -21600.002} C_VEL
LIN {X 0,Y 199.995,Z 173.563,A -85,B 0,C 180,E1 -21604.032,E2 -21604.032} C_VEL
LIN {X 0,Y 200.078,Z 173.557,A -85,B 0,C 180,E1 -21608.079,E2 -21608.079} C_VEL
LIN {X 0,Y 199.865,Z 173.573,A -85,B 0,C 180,E1 -21612.182,E2 -21612.182} C_VEL
LIN {X 0,Y 199.762,Z 173.584,A -85,B 0,C 180,E1 -21616.349,E2 -21616.349} C_VEL
LIN {X 0,Y 199.648,Z 173.603,A -85,B 0,C 180,E1 -21620.613,E2 -21620.613} C_VEL
LIN {X 0,Y 199.637,Z 173.608,A -85,B 0,C 180,E1 -21624.991,E2 -21624.991} C_VEL
LIN {X 0,Y 199.61,Z 173.612,A -85,B 0,C 180,E1 -21629.534,E2 -21629.534} C_VEL
LIN {X 0,Y 199.668,Z 173.613,A -85,B 0,C 180,E1 -21632.354,E2 -21632.354} C_VEL
LIN {X 0,Y 199.627,Z 173.809,A -85,B 0,C 180,E1 -21636.258,E2 -21636.258} C_VEL
LIN {X 0,Y 201.353,Z 179.1,A -85,B 0,C 180,E1 -21640.549,E2 -21640.549} C_VEL
LIN {X 0,Y 204.34,Z 183.66,A -85,B 0,C 180,E1 -21642.048,E2 -21642.048} C_VEL
LIN {X 0,Y 206.114,Z 186.116,A -85,B 0,C 180,E1 -21642.876,E2 -21642.876} C_VEL
LIN {X 0,Y 210.028,Z 192.291,A -85,B 0,C 180,E1 -21644.646,E2 -21644.646} C_VEL
LIN {X 0,Y 213.297,Z 197.789,A -85,B 0,C 180,E1 -21646.035,E2 -21646.035} C_VEL
LIN {X 0,Y 217.288,Z 204.59,A -85,B 0,C 180,E1 -21647.611,E2 -21647.611} C_VEL
LIN {X 0,Y 219.473,Z 209.044,A -85,B 0,C 180,E1 -21648.457,E2 -21648.457} C_VEL
LIN {X 0,Y 221.033,Z 214.156,A -85,B 0,C 180,E1 -21649.136,E2 -21649.136} C_VEL
LIN {X 0,Y 221.798,Z 217.773,A -85,B 0,C 180,E1 -21649.515,E2 -21649.515} C_VEL
LIN {X 0,Y 223.911,Z 233.113,A -85,B 0,C 180,E1 -21650.784,E2 -21650.784} C_VEL
LIN {X 0,Y 224.942,Z 243.535,A -85,B 0,C 180,E1 -21651.519,E2 -21651.519} C_VEL
LIN {X 0,Y 222.08,Z 290.167,A -85,B 0,C 180,E1 -21653.039,E2 -21653.039} C_VEL
LIN {X 0,Y 220.273,Z 304.17,A -85,B 0,C 180,E1 -21653.825,E2 -21653.825} C_VEL
LIN {X 0,Y 217.913,Z 316.14,A -85,B 0,C 180,E1 -21654.796,E2 -21654.796} C_VEL
LIN {X 0,Y 214.741,Z 328.603,A -85,B 0,C 180,E1 -21656.195,E2 -21656.195} C_VEL
LIN {X 0,Y 211.567,Z 339.739,A -85,B 0,C 180,E1 -21657.893,E2 -21657.893} C_VEL
LIN {X 0,Y 208.128,Z 349.834,A -85,B 0,C 180,E1 -21659.848,E2 -21659.848} C_VEL
LIN {X 0,Y 204.25,Z 359.779,A -85,B 0,C 180,E1 -21662.321,E2 -21662.321} C_VEL
LIN {X 0,Y 200.686,Z 368.567,A -85,B 0,C 180,E1 -21665.151,E2 -21665.151} C_VEL
LIN {X 0,Y 197.736,Z 375.631,A -85,B 0,C 180,E1 -21668.088,E2 -21668.088} C_VEL
LIN {X 0,Y 195.144,Z 381.31,A -85,B 0,C 180,E1 -21671.087,E2 -21671.087} C_VEL
LIN {X 0,Y 193.002,Z 385.81,A -85,B 0,C 180,E1 -21674.151,E2 -21674.151} C_VEL
LIN {X 0,Y 191.601,Z 389.256,A -85,B 0,C 180,E1 -21677.287,E2 -21677.287} C_VEL
LIN {X 0,Y 190.476,Z 392.324,A -85,B 0,C 180,E1 -21681.513,E2 -21681.513} C_VEL
LIN {X 0,Y 190.228,Z 393.27,A -85,B 0,C 180,E1 -21683.637,E2 -21683.637} C_VEL
LIN {X 0,Y 190.173,Z 393.846,A -85,B 0,C 180,E1 -21686.226,E2 -21686.226} C_VEL
LIN {X 0,Y 190.386,Z 393.645,A -85,B 0,C 180,E1 -21690,E2 -21690} C_VEL
LIN {X 0,Y 190.18,Z 392.117,A -85,B 0,C 180,E1 -21693.805,E2 -21693.805} C_VEL
LIN {X 0,Y 190.281,Z 390.306,A -85,B 0,C 180,E1 -21696.362,E2 -21696.362} C_VEL
LIN {X 0,Y 190.688,Z 387.158,A -85,B 0,C 180,E1 -21699.547,E2 -21699.547} C_VEL
LIN {X 0,Y 191.488,Z 382.92,A -85,B 0,C 180,E1 -21702.722,E2 -21702.722} C_VEL
LIN {X 0,Y 193.117,Z 376.462,A -85,B 0,C 180,E1 -21706.383,E2 -21706.383} C_VEL
LIN {X 0,Y 195.107,Z 369.393,A -85,B 0,C 180,E1 -21709.463,E2 -21709.463} C_VEL
LIN {X 0,Y 197.107,Z 361.724,A -85,B 0,C 180,E1 -21712.129,E2 -21712.129} C_VEL
LIN {X 0,Y 199.326,Z 353.368,A -85,B 0,C 180,E1 -21714.475,E2 -21714.475} C_VEL
LIN {X 0,Y 202.085,Z 342.565,A -85,B 0,C 180,E1 -21716.88,E2 -21716.88} C_VEL
LIN {X 0,Y 204.628,Z 331.814,A -85,B 0,C 180,E1 -21718.741,E2 -21718.741} C_VEL
LIN {X 0,Y 207.033,Z 319.761,A -85,B 0,C 180,E1 -21720.329,E2 -21720.329} C_VEL
LIN {X 0,Y 209.077,Z 307.25,A -85,B 0,C 180,E1 -21721.543,E2 -21721.543} C_VEL
LIN {X 0,Y 210.519,Z 294.165,A -85,B 0,C 180,E1 -21722.427,E2 -21722.427} C_VEL
LIN {X 0,Y 211.534,Z 277.16,A -85,B 0,C 180,E1 -21723.091,E2 -21723.091} C_VEL
LIN {X 0,Y 213.147,Z 239.517,A -85,B 0,C 180,E1 -21724.351,E2 -21724.351} C_VEL
LIN {X 0,Y 210.469,Z 218.686,A -85,B 0,C 180,E1 -21725.619,E2 -21725.619} C_VEL
LIN {X 0,Y 203.411,Z 200.7,A -85,B 0,C 180,E1 -21727.577,E2 -21727.577} C_VEL
LIN {X 0,Y 197.594,Z 188.15,A -85,B 0,C 180,E1 -21729.219,E2 -21729.219} C_VEL
LIN {X 0,Y 194.152,Z 180.902,A -85,B 0,C 180,E1 -21730.319,E2 -21730.319} C_VEL
LIN {X 0,Y 192.529,Z 174.499,A -85,B 0,C 180,E1 -21733.914,E2 -21733.914} C_VEL
LIN {X 0,Y 192.509,Z 174.508,A -85,B 0,C 180,E1 -21738.916,E2 -21738.916} C_VEL
LIN {X 0,Y 192.587,Z 174.5,A -85,B 0,C 180,E1 -21743.403,E2 -21743.403} C_VEL
LIN {X 0,Y 192.61,Z 174.497,A -85,B 0,C 180,E1 -21747.06,E2 -21747.06} C_VEL
LIN {X 0,Y 192.626,Z 174.491,A -85,B 0,C 180,E1 -21751.684,E2 -21751.684} C_VEL
LIN {X 0,Y 192.676,Z 174.485,A -85,B 0,C 180,E1 -21756.343,E2 -21756.343} C_VEL
LIN {X 0,Y 192.699,Z 174.48,A -85,B 0,C 180,E1 -21761.49,E2 -21761.49} C_VEL
LIN {X 0,Y 192.726,Z 174.477,A -85,B 0,C 180,E1 -21765.209,E2 -21765.209} C_VEL
LIN {X 0,Y 192.949,Z 174.439,A -85,B 0,C 180,E1 -21769.565,E2 -21769.565} C_VEL
LIN {X 0,Y 192.97,Z 174.431,A -85,B 0,C 180,E1 -21773.726,E2 -21773.726} C_VEL
LIN {X 0,Y 193.234,Z 174.415,A -85,B 0,C 180,E1 -21777.914,E2 -21777.914} C_VEL
LIN {X 0,Y 193.418,Z 174.384,A -85,B 0,C 180,E1 -21779.998,E2 -21779.998} C_VEL
LIN {X 0,Y 192.937,Z 174.422,A -85,B 0,C 180,E1 -21784.176,E2 -21784.176} C_VEL
LIN {X 0,Y 193.028,Z 174.44,A -85,B 0,C 180,E1 -21788.372,E2 -21788.372} C_VEL
LIN {X 0,Y 192.775,Z 174.462,A -85,B 0,C 180,E1 -21792.633,E2 -21792.633} C_VEL
LIN {X 0,Y 192.695,Z 174.47,A -85,B 0,C 180,E1 -21798.506,E2 -21798.506} C_VEL
LIN {X 0,Y 192.619,Z 174.483,A -85,B 0,C 180,E1 -21804.192,E2 -21804.192} C_VEL
LIN {X 0,Y 192.599,Z 174.473,A -85,B 0,C 180,E1 -21808.863,E2 -21808.863} C_VEL
LIN {X 0,Y 192.593,Z 174.496,A -85,B 0,C 180,E1 -21813.185,E2 -21813.185} C_VEL
LIN {X 0,Y 192.538,Z 174.477,A -85,B 0,C 180,E1 -21818.353,E2 -21818.353} C_VEL
LIN {X 0,Y 192.482,Z 174.512,A -85,B 0,C 180,E1 -21823.092,E2 -21823.092} C_VEL
LIN {X 0,Y 192.48,Z 174.493,A -85,B 0,C 180,E1 -21826.905,E2 -21826.905} C_VEL
LIN {X 0,Y 192.538,Z 174.505,A -85,B 0,C 180,E1 -21831.644,E2 -21831.644} C_VEL
LIN {X 0,Y 192.59,Z 174.492,A -85,B 0,C 180,E1 -21836.812,E2 -21836.812} C_VEL
LIN {X 0,Y 192.614,Z 174.483,A -85,B 0,C 180,E1 -21841.683,E2 -21841.683} C_VEL
LIN {X 0,Y 192.652,Z 174.474,A -85,B 0,C 180,E1 -21846.341,E2 -21846.341} C_VEL
LIN {X 0,Y 192.734,Z 174.663,A -85,B 0,C 180,E1 -21851.775,E2 -21851.775} C_VEL
LIN {X 0,Y 193.731,Z 177.395,A -85,B 0,C 180,E1 -21852.109,E2 -21852.109} C_VEL
LIN {X 0,Y 195.184,Z 179.558,A -85,B 0,C 180,E1 -21852.508,E2 -21852.508} C_VEL
LIN {X 0,Y 204.624,Z 196.271,A -85,B 0,C 180,E1 -21855.054,E2 -21855.054} C_VEL
LIN {X 0,Y 209.448,Z 205.913,A -85,B 0,C 180,E1 -21856.287,E2 -21856.287} C_VEL
LIN {X 0,Y 214.201,Z 218.676,A -85,B 0,C 180,E1 -21857.577,E2 -21857.577} C_VEL
LIN {X 0,Y 211.159,Z 277.137,A -85,B 0,C 180,E1 -21859.52,E2 -21859.52} C_VEL
LIN {X 0,Y 209.838,Z 290.783,A -85,B 0,C 180,E1 -21860.359,E2 -21860.359} C_VEL
LIN {X 0,Y 208.271,Z 303.14,A -85,B 0,C 180,E1 -21861.51,E2 -21861.51} C_VEL
LIN {X 0,Y 206.13,Z 315.763,A -85,B 0,C 180,E1 -21863.124,E2 -21863.124} C_VEL
LIN {X 0,Y 203.701,Z 327.322,A -85,B 0,C 180,E1 -21865.051,E2 -21865.051} C_VEL
LIN {X 0,Y 201.187,Z 337.563,A -85,B 0,C 180,E1 -21867.246,E2 -21867.246} C_VEL
LIN {X 0,Y 198.557,Z 347.644,A -85,B 0,C 180,E1 -21870,E2 -21870} C_VEL
LIN {X 0,Y 196.4,Z 355.144,A -85,B 0,C 180,E1 -21872.563,E2 -21872.563} C_VEL
LIN {X 0,Y 194.283,Z 362.457,A -85,B 0,C 180,E1 -21875.709,E2 -21875.709} C_VEL
LIN {X 0,Y 192.899,Z 367.411,A -85,B 0,C 180,E1 -21878.379,E2 -21878.379} C_VEL
LIN {X 0,Y 191.593,Z 372.155,A -85,B 0,C 180,E1 -21881.639,E2 -21881.639} C_VEL
LIN {X 0,Y 190.654,Z 375.744,A -85,B 0,C 180,E1 -21884.953,E2 -21884.953} C_VEL
LIN {X 0,Y 190.257,Z 377.522,A -85,B 0,C 180,E1 -21887.188,E2 -21887.188} C_VEL
LIN {X 0,Y 189.999,Z 378.87,A -85,B 0,C 180,E1 -21889.445,E2 -21889.445} C_VEL
LIN {X 0,Y 189.969,Z 379.884,A -85,B 0,C 180,E1 -21892.354,E2 -21892.354} C_VEL
LIN {X 0,Y 190.283,Z 380.116,A -85,B 0,C 180,E1 -21896.309,E2 -21896.309} C_VEL
LIN {X 0,Y 190.715,Z 379.587,A -85,B 0,C 180,E1 -21898.624,E2 -21898.624} C_VEL
LIN {X 0,Y 191.996,Z 377.526,A -85,B 0,C 180,E1 -21902.661,E2 -21902.661} C_VEL
LIN {X 0,Y 193.301,Z 375.072,A -85,B 0,C 180,E1 -21905.572,E2 -21905.572} C_VEL
LIN {X 0,Y 195.422,Z 370.992,A -85,B 0,C 180,E1 -21909.002,E2 -21909.002} C_VEL
LIN {X 0,Y 198.083,Z 365.515,A -85,B 0,C 180,E1 -21912.386,E2 -21912.386} C_VEL
LIN {X 0,Y 200.882,Z 359.581,A -85,B 0,C 180,E1 -21915.18,E2 -21915.18} C_VEL
LIN {X 0,Y 203.97,Z 352.548,A -85,B 0,C 180,E1 -21917.8,E2 -21917.8} C_VEL
LIN {X 0,Y 207.216,Z 344.418,A -85,B 0,C 180,E1 -21920.215,E2 -21920.215} C_VEL
LIN {X 0,Y 210.999,Z 333.85,A -85,B 0,C 180,E1 -21922.677,E2 -21922.677} C_VEL
LIN {X 0,Y 214.093,Z 324.064,A -85,B 0,C 180,E1 -21924.452,E2 -21924.452} C_VEL
LIN {X 0,Y 217.069,Z 312.735,A -85,B 0,C 180,E1 -21926.063,E2 -21926.063} C_VEL
LIN {X 0,Y 219.638,Z 300.424,A -85,B 0,C 180,E1 -21927.393,E2 -21927.393} C_VEL
LIN {X 0,Y 221.603,Z 287.339,A -85,B 0,C 180,E1 -21928.422,E2 -21928.422} C_VEL
LIN {X 0,Y 222.874,Z 275.299,A -85,B 0,C 180,E1 -21929.017,E2 -21929.017} C_VEL
LIN {X 0,Y 225.717,Z 227.329,A -85,B 0,C 180,E1 -21930.551,E2 -21930.551} C_VEL
LIN {X 0,Y 220.696,Z 216.096,A -85,B 0,C 180,E1 -21932.375,E2 -21932.375} C_VEL
LIN {X 0,Y 216.41,Z 208.182,A -85,B 0,C 180,E1 -21933.984,E2 -21933.984} C_VEL
LIN {X 0,Y 209.701,Z 197.801,A -85,B 0,C 180,E1 -21936.665,E2 -21936.665} C_VEL
LIN {X 0,Y 206.443,Z 193.241,A -85,B 0,C 180,E1 -21938.084,E2 -21938.084} C_VEL
LIN {X 0,Y 203.717,Z 189.492,A -85,B 0,C 180,E1 -21939.343,E2 -21939.343} C_VEL
LIN {X 0,Y 201.068,Z 185.935,A -85,B 0,C 180,E1 -21940.634,E2 -21940.634} C_VEL
LIN {X 0,Y 200.271,Z 184.858,A -85,B 0,C 180,E1 -21941.044,E2 -21941.044} C_VEL
LIN {X 0,Y 197.864,Z 182.074,A -85,B 0,C 180,E1 -21942.308,E2 -21942.308} C_VEL
LIN {X 0,Y 196.749,Z 179.99,A -85,B 0,C 180,E1 -21942.983,E2 -21942.983} C_VEL
LIN {X 0,Y 194.21,Z 177.995,A -85,B 0,C 180,E1 -21944.388,E2 -21944.388} C_VEL
LIN {X 0,Y 192.967,Z 175.534,A -85,B 0,C 180,E1 -21945.232,E2 -21945.232} C_VEL
LIN {X 0,Y 192.781,Z 174.465,A -85,B 0,C 180,E1 -21945.487,E2 -21945.487} C_VEL
LIN {X 0,Y 192.945,Z 174.445,A -85,B 0,C 180,E1 -21949.568,E2 -21949.568} C_VEL
LIN {X 0,Y 192.974,Z 174.444,A -85,B 0,C 180,E1 -21953.729,E2 -21953.729} C_VEL
LIN {X 0,Y 193.258,Z 174.406,A -85,B 0,C 180,E1 -21957.918,E2 -21957.918} C_VEL
LIN {X 0,Y 193.432,Z 174.37,A -85,B 0,C 180,E1 -21960.002,E2 -21960.002} C_VEL
LIN {X 0,Y 192.942,Z 174.439,A -85,B 0,C 180,E1 -21964.179,E2 -21964.179} C_VEL
LIN {X 0,Y 193.029,Z 174.437,A -85,B 0,C 180,E1 -21968.376,E2 -21968.376} C_VEL
LIN {X 0,Y 192.791,Z 174.458,A -85,B 0,C 180,E1 -21972.636,E2 -21972.636} C_VEL
LIN {X 0,Y 192.716,Z 174.462,A -85,B 0,C 180,E1 -21976.964,E2 -21976.964} C_VEL
LIN {X 0,Y 192.581,Z 174.48,A -85,B 0,C 180,E1 -21981.405,E2 -21981.405} C_VEL
LIN {X 0,Y 192.628,Z 174.49,A -85,B 0,C 180,E1 -21984.2,E2 -21984.2} C_VEL
LIN {X 0,Y 192.603,Z 174.491,A -85,B 0,C 180,E1 -21988.867,E2 -21988.867} C_VEL
LIN {X 0,Y 192.581,Z 174.601,A -85,B 0,C 180,E1 -21993.347,E2 -21993.347} C_VEL
LIN {X 0,Y 193.899,Z 178.571,A -85,B 0,C 180,E1 -21997.01,E2 -21997.01} C_VEL
LIN {X 0,Y 197.094,Z 183.315,A -85,B 0,C 180,E1 -21998.94,E2 -21998.94} C_VEL
LIN {X 0,Y 198.678,Z 185.352,A -85,B 0,C 180,E1 -21999.81,E2 -21999.81} C_VEL
LIN {X 0,Y 203.124,Z 192.041,A -85,B 0,C 180,E1 -22002.101,E2 -22002.101} C_VEL
LIN {X 0,Y 206.731,Z 197.813,A -85,B 0,C 180,E1 -22003.809,E2 -22003.809} C_VEL
LIN {X 0,Y 210.447,Z 204.245,A -85,B 0,C 180,E1 -22005.468,E2 -22005.468} C_VEL
LIN {X 0,Y 214.328,Z 211.184,A -85,B 0,C 180,E1 -22007.068,E2 -22007.068} C_VEL
LIN {X 0,Y 219.522,Z 222.065,A -85,B 0,C 180,E1 -22009.116,E2 -22009.116} C_VEL
LIN {X 0,Y 223.911,Z 233.113,A -85,B 0,C 180,E1 -22010.784,E2 -22010.784} C_VEL
LIN {X 0,Y 224.09,Z 236.924,A -85,B 0,C 180,E1 -22011.005,E2 -22011.005} C_VEL
LIN {X 0,Y 223.387,Z 242.782,A -85,B 0,C 180,E1 -22011.102,E2 -22011.102} C_VEL
LIN {X 0,Y 219.882,Z 256.454,A -85,B 0,C 180,E1 -22010.862,E2 -22010.862} C_VEL
LIN {X 0,Y 218.766,Z 262.426,A -85,B 0,C 180,E1 -22010.861,E2 -22010.861} C_VEL
LIN {X 0,Y 218.586,Z 264.433,A -85,B 0,C 180,E1 -22010.91,E2 -22010.91} C_VEL
LIN {X 0,Y 216.827,Z 290.459,A -85,B 0,C 180,E1 -22011.8,E2 -22011.8} C_VEL
LIN {X 0,Y 215.002,Z 303.929,A -85,B 0,C 180,E1 -22012.57,E2 -22012.57} C_VEL
LIN {X 0,Y 212.646,Z 315.378,A -85,B 0,C 180,E1 -22013.495,E2 -22013.495} C_VEL
LIN {X 0,Y 209.859,Z 326.358,A -85,B 0,C 180,E1 -22014.712,E2 -22014.712} C_VEL
LIN {X 0,Y 206.453,Z 337.835,A -85,B 0,C 180,E1 -22016.415,E2 -22016.415} C_VEL
LIN {X 0,Y 202.802,Z 348.221,A -85,B 0,C 180,E1 -22018.389,E2 -22018.389} C_VEL
LIN {X 0,Y 199.418,Z 356.746,A -85,B 0,C 180,E1 -22020.436,E2 -22020.436} C_VEL
LIN {X 0,Y 196.041,Z 364.649,A -85,B 0,C 180,E1 -22022.801,E2 -22022.801} C_VEL
LIN {X 0,Y 192.529,Z 372.642,A -85,B 0,C 180,E1 -22025.869,E2 -22025.869} C_VEL
LIN {X 0,Y 190.135,Z 377.742,A -85,B 0,C 180,E1 -22028.307,E2 -22028.307} C_VEL
LIN {X 0,Y 187.598,Z 382.95,A -85,B 0,C 180,E1 -22031.432,E2 -22031.432} C_VEL
LIN {X 0,Y 185.535,Z 387.02,A -85,B 0,C 180,E1 -22034.624,E2 -22034.624} C_VEL
LIN {X 0,Y 184.642,Z 389.145,A -85,B 0,C 180,E1 -22036.799,E2 -22036.799} C_VEL
LIN {X 0,Y 183.43,Z 392.153,A -85,B 0,C 180,E1 -22041.185,E2 -22041.185} C_VEL
LIN {X 0,Y 183.145,Z 393.067,A -85,B 0,C 180,E1 -22043.39,E2 -22043.39} C_VEL
LIN {X 0,Y 183.085,Z 393.633,A -85,B 0,C 180,E1 -22046.444,E2 -22046.444} C_VEL
LIN {X 0,Y 183.304,Z 393.348,A -85,B 0,C 180,E1 -22050,E2 -22050} C_VEL
LIN {X 0,Y 183.101,Z 391.933,A -85,B 0,C 180,E1 -22053.632,E2 -22053.632} C_VEL
LIN {X 0,Y 183.317,Z 388.973,A -85,B 0,C 180,E1 -22057.712,E2 -22057.712} C_VEL
LIN {X 0,Y 183.886,Z 385.418,A -85,B 0,C 180,E1 -22061.017,E2 -22061.017} C_VEL
LIN {X 0,Y 184.894,Z 380.726,A -85,B 0,C 180,E1 -22064.305,E2 -22064.305} C_VEL
LIN {X 0,Y 186.941,Z 373.648,A -85,B 0,C 180,E1 -22068.069,E2 -22068.069} C_VEL
LIN {X 0,Y 189.135,Z 365.953,A -85,B 0,C 180,E1 -22071.242,E2 -22071.242} C_VEL
LIN {X 0,Y 191.293,Z 358.048,A -85,B 0,C 180,E1 -22073.838,E2 -22073.838} C_VEL
LIN {X 0,Y 193.934,Z 348.397,A -85,B 0,C 180,E1 -22076.356,E2 -22076.356} C_VEL
LIN {X 0,Y 196.703,Z 337.703,A -85,B 0,C 180,E1 -22078.547,E2 -22078.547} C_VEL
LIN {X 0,Y 199.095,Z 327.388,A -85,B 0,C 180,E1 -22080.201,E2 -22080.201} C_VEL
LIN {X 0,Y 201.481,Z 315.113,A -85,B 0,C 180,E1 -22081.696,E2 -22081.696} C_VEL
LIN {X 0,Y 203.363,Z 302.246,A -85,B 0,C 180,E1 -22082.83,E2 -22082.83} C_VEL
LIN {X 0,Y 204.668,Z 289.567,A -85,B 0,C 180,E1 -22083.574,E2 -22083.574} C_VEL
LIN {X 0,Y 206.968,Z 240.053,A -85,B 0,C 180,E1 -22085.308,E2 -22085.308} C_VEL
LIN {X 0,Y 204.612,Z 221.23,A -85,B 0,C 180,E1 -22086.488,E2 -22086.488} C_VEL
LIN {X 0,Y 197.79,Z 203.759,A -85,B 0,C 180,E1 -22088.477,E2 -22088.477} C_VEL
LIN {X 0,Y 191.101,Z 189.254,A -85,B 0,C 180,E1 -22090.486,E2 -22090.486} C_VEL
LIN {X 0,Y 186.834,Z 180.69,A -85,B 0,C 180,E1 -22091.847,E2 -22091.847} C_VEL
LIN {X 0,Y 185.45,Z 175.385,A -85,B 0,C 180,E1 -22095.028,E2 -22095.028} C_VEL
LIN {X 0,Y 185.461,Z 175.387,A -85,B 0,C 180,E1 -22099.891,E2 -22099.891} C_VEL
LIN {X 0,Y 185.505,Z 175.381,A -85,B 0,C 180,E1 -22102.713,E2 -22102.713} C_VEL
LIN {X 0,Y 185.536,Z 175.375,A -85,B 0,C 180,E1 -22107.972,E2 -22107.972} C_VEL
LIN {X 0,Y 185.552,Z 175.373,A -85,B 0,C 180,E1 -22110.594,E2 -22110.594} C_VEL
LIN {X 0,Y 185.585,Z 175.368,A -85,B 0,C 180,E1 -22115.38,E2 -22115.38} C_VEL
LIN {X 0,Y 185.63,Z 175.362,A -85,B 0,C 180,E1 -22121.177,E2 -22121.177} C_VEL
LIN {X 0,Y 185.712,Z 175.352,A -85,B 0,C 180,E1 -22126.874,E2 -22126.874} C_VEL
LIN {X 0,Y 185.978,Z 175.292,A -85,B 0,C 180,E1 -22131.304,E2 -22131.304} C_VEL
LIN {X 0,Y 186.18,Z 175.294,A -85,B 0,C 180,E1 -22137.835,E2 -22137.835} C_VEL
LIN {X 0,Y 186.383,Z 175.26,A -85,B 0,C 180,E1 -22139.998,E2 -22139.998} C_VEL
LIN {X 0,Y 185.885,Z 175.299,A -85,B 0,C 180,E1 -22144.335,E2 -22144.335} C_VEL
LIN {X 0,Y 185.977,Z 175.318,A -85,B 0,C 180,E1 -22148.692,E2 -22148.692} C_VEL
